KUKA KRL program: MyProgram_206().src

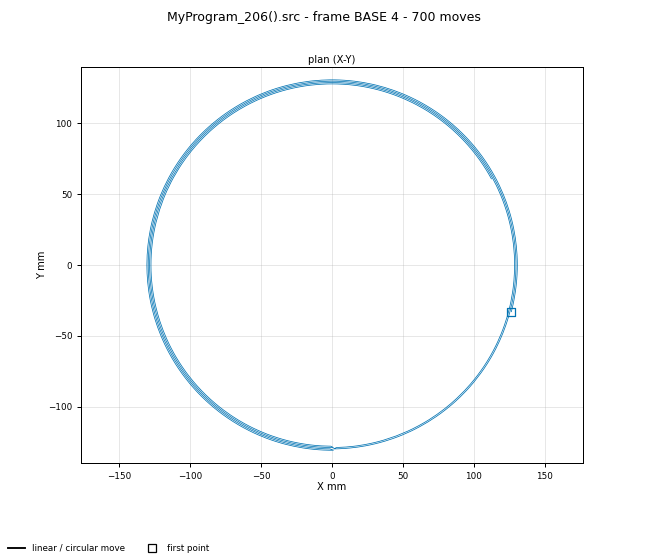
[picture p0: tool path of MyProgram_206().src in frame BASE 4, 700 of 700 moves have a stored position in this frame; points joined in program order, loops and branches not executed]
&ACCESS RVP
&REL 1
&PARAM TEMPLATE = C:\KRC\Roboter\Template\vorgabe
&PARAM EDITMASK = *
DEF MyProgram_206()
; ---- Setting reference (Base) ----
$BASE = BASE_DATA[4]

; --------------------------
; ---- Setting tool (TCP) ----
$TOOL = TOOL_DATA[3]
; --------------------------

$VEL.CP = VEL_APROX_PRINT
Startdeposition()
$VEL.CP = VEL_PRINT
LIN {X 126.4468,Y -32.9033,Z 147,A -17.6105,B 24.9579,C -1.4995,E1 25.155,E2 463.9583} C_DIS
LIN {X 127.5485,Y -28.3334,Z 147,A -15.6439,B 24.9578,C -1.501,E1 25.1563,E2 461.9995} C_DIS
LIN {X 128.2452,Y -24.9837,Z 147,A -14.1957,B 24.9577,C -1.5031,E1 25.1571,E2 460.5549} C_DIS
LIN {X 128.8355,Y -21.7323,Z 147,A -12.7991,B 24.9576,C -1.505,E1 25.1577,E2 459.162} C_DIS
LIN {X 129.3075,Y -18.7203,Z 147,A -11.4837,B 24.9574,C -1.5082,E1 25.1583,E2 457.8467} C_DIS
LIN {X 129.825,Y -14.7267,Z 147,A -9.5964,B 24.9567,C -1.5207,E1 25.1589,E2 455.9413} C_DIS
LIN {X 130.2553,Y -10.2444,Z 147,A -7.7715,B 24.9567,C -1.519,E1 25.1594,E2 454.1311} C_DIS
LIN {X 130.4729,Y -6.9157,Z 147,A -6.2379,B 24.9563,C -1.5277,E1 25.1596,E2 452.586} C_DIS
LIN {X 130.6151,Y -3.2719,Z 147,A -4.7193,B 24.9563,C -1.5286,E1 25.1598,E2 451.0743} C_DIS
LIN {X 130.6591,Y 0,Z 147,A -3.1934,B 24.9557,C -1.5383,E1 25.1598,E2 449.5347} C_DIS
LIN {X 130.6081,Y 3.5243,Z 147,A -1.7202,B 24.9556,C -1.5395,E1 25.1597,E2 448.0675} C_DIS
LIN {X 130.4538,Y 7.2957,Z 147,A 0.0234,B 24.955,C -1.5497,E1 25.1595,E2 446.3101} C_DIS
LIN {X 130.1886,Y 11.036,Z 147,A 1.3411,B 24.9557,C -1.5373,E1 25.1592,E2 445.0295} C_DIS
LIN {X 129.9628,Y 13.4458,Z 147,A 2.6602,B 24.9547,C -1.5548,E1 25.1588,E2 443.6769} C_DIS
LIN {X 129.6461,Y 16.2263,Z 147,A 3.8628,B 24.9546,C -1.5574,E1 25.1584,E2 442.4753} C_DIS
LIN {X 129.2338,Y 19.2365,Z 147,A 5.1142,B 24.9546,C -1.5574,E1 25.1579,E2 441.2315} C_DIS
LIN {X 128.6452,Y 22.8309,Z 147,A 6.4775,B 24.955,C -1.5498,E1 25.1573,E2 439.8941} C_DIS
LIN {X 128.1418,Y 25.5106,Z 147,A 7.8931,B 24.9541,C -1.5656,E1 25.1565,E2 438.4495} C_DIS
LIN {X 127.5485,Y 28.3334,Z 147,A 9.2267,B 24.9536,C -1.5733,E1 25.1557,E2 437.1054} C_DIS
LIN {X 126.7277,Y 31.7964,Z 147,A 10.7556,B 24.9534,C -1.5765,E1 25.1547,E2 435.5777} C_DIS
LIN {X 125.9076,Y 34.9019,Z 147,A 12.104,B 24.9534,C -1.5777,E1 25.1537,E2 434.2343} C_DIS
LIN {X 124.9889,Y 38.0602,Z 147,A 13.541,B 24.9531,C -1.5819,E1 25.1526,E2 432.7957} C_DIS
LIN {X 123.9957,Y 41.1807,Z 147,A 14.8652,B 24.9532,C -1.5802,E1 25.1515,E2 431.4829} C_DIS
LIN {X 122.993,Y 44.0856,Z 147,A 16.2938,B 24.9527,C -1.5887,E1 25.1501,E2 430.0423} C_DIS
LIN {X 121.8877,Y 47.0557,Z 147,A 17.4959,B 24.9531,C -1.5827,E1 25.149,E2 428.861} C_DIS
LIN {X 120.8768,Y 49.6004,Z 147,A 18.8871,B 24.9522,C -1.5966,E1 25.1475,E2 427.4448} C_DIS
LIN {X 119.4073,Y 53.0353,Z 147,A 20.3317,B 24.9526,C -1.5909,E1 25.1459,E2 426.0214} C_DIS
LIN {X 118.1445,Y 55.7938,Z 147,A 21.9257,B 24.9515,C -1.6091,E1 25.144,E2 424.3933} C_DIS
LIN {X 116.5299,Y 59.0893,Z 147,A 23.3217,B 24.9519,C -1.6022,E1 25.1423,E2 423.021} C_DIS
LIN {X 114.9008,Y 62.2029,Z 147,A 25.1201,B 24.9508,C -1.6204,E1 25.1399,E2 421.1891} C_DIS
LIN {X 112.8073,Y 65.923,Z 147,A 26.8375,B 24.951,C -1.6172,E1 25.1375,E2 419.4881} C_DIS
LIN {X 110.7749,Y 69.2838,Z 147,A 28.6456,B 24.9504,C -1.6265,E1 25.1348,E2 417.6673} C_DIS
LIN {X 108.4346,Y 72.8927,Z 147,A 30.56,B 24.95,C -1.633,E1 25.1319,E2 415.7472} C_DIS
LIN {X 105.9386,Y 76.4742,Z 147,A 32.4107,B 24.95,C -1.6345,E1 25.1289,E2 413.9019} C_DIS
LIN {X 103.4746,Y 79.7768,Z 147,A 34.2161,B 24.9497,C -1.6389,E1 25.1258,E2 412.0946} C_DIS
LIN {X 100.8929,Y 83.0182,Z 147,A 36.0737,B 24.9493,C -1.6455,E1 25.1226,E2 410.2301} C_DIS
LIN {X 97.9836,Y 86.4318,Z 147,A 37.9938,B 24.9491,C -1.6476,E1 25.1191,E2 408.3137} C_DIS
LIN {X 94.9376,Y 89.767,Z 147,A 39.9231,B 24.9491,C -1.6494,E1 25.1154,E2 406.3886} C_DIS
LIN {X 91.9122,Y 92.8625,Z 147,A 41.8417,B 24.9487,C -1.6547,E1 25.1116,E2 404.4657} C_DIS
LIN {X 88.7329,Y 95.9056,Z 147,A 43.8155,B 24.9483,C -1.6611,E1 25.1076,E2 402.485} C_DIS
LIN {X 85.5245,Y 98.777,Z 147,A 45.651,B 24.9483,C -1.6621,E1 25.1037,E2 400.6542} C_DIS
LIN {X 82.3328,Y 101.4529,Z 147,A 47.4623,B 24.9481,C -1.6649,E1 25.0998,E2 398.8434} C_DIS
LIN {X 79.0403,Y 104.0387,Z 147,A 49.2387,B 24.9481,C -1.6651,E1 25.0959,E2 397.0729} C_DIS
LIN {X 76.2379,Y 106.109,Z 147,A 50.8439,B 24.9476,C -1.6719,E1 25.0923,E2 395.4573} C_DIS
LIN {X 72.8927,Y 108.4346,Z 147,A 52.6181,B 24.9475,C -1.6743,E1 25.0882,E2 393.6835} C_DIS
LIN {X 69.2662,Y 110.7858,Z 147,A 54.5215,B 24.9473,C -1.6778,E1 25.0837,E2 391.778} C_DIS
LIN {X 65.2644,Y 113.1894,Z 147,A 56.5241,B 24.9473,C -1.6785,E1 25.0789,E2 389.7798} C_DIS
LIN {X 61.4738,Y 115.2926,Z 147,A 58.3276,B 24.9473,C -1.676,E1 25.0745,E2 387.9873} C_DIS
LIN {X 58.5401,Y 116.8095,Z 147,A 59.7705,B 24.9473,C -1.6777,E1 25.0709,E2 386.5445} C_DIS
LIN {X 55.1242,Y 118.4574,Z 147,A 61.4114,B 24.9472,C -1.6786,E1 25.0668,E2 384.9056} C_DIS
LIN {X 52.3074,Y 119.7285,Z 147,A 62.8038,B 24.947,C -1.6821,E1 25.0632,E2 383.5084} C_DIS
LIN {X 49.2079,Y 121.0351,Z 147,A 64.186,B 24.9472,C -1.6789,E1 25.0597,E2 382.1371} C_DIS
LIN {X 46.0827,Y 122.2588,Z 147,A 65.7194,B 24.9469,C -1.6835,E1 25.0557,E2 380.5959} C_DIS
LIN {X 43.1226,Y 123.3342,Z 147,A 67.0966,B 24.9469,C -1.6846,E1 25.052,E2 379.2191} C_DIS
LIN {X 40.044,Y 124.3678,Z 147,A 68.3559,B 24.9473,C -1.6773,E1 25.0487,E2 377.9794} C_DIS
LIN {X 37.0878,Y 125.2814,Z 147,A 69.887,B 24.9466,C -1.6873,E1 25.0446,E2 376.4274} C_DIS
LIN {X 34.0705,Y 126.1355,Z 147,A 71.0918,B 24.9471,C -1.6795,E1 25.0414,E2 375.243} C_DIS
LIN {X 31.1608,Y 126.8862,Z 147,A 72.5499,B 24.9466,C -1.6875,E1 25.0374,E2 373.7681} C_DIS
LIN {X 28.3334,Y 127.5485,Z 147,A 73.8201,B 24.9466,C -1.688,E1 25.034,E2 372.4985} C_DIS
LIN {X 24.8107,Y 128.2783,Z 147,A 75.2022,B 24.9472,C -1.6788,E1 25.0302,E2 371.14} C_DIS
LIN {X 22.0424,Y 128.7837,Z 147,A 76.6946,B 24.9463,C -1.6924,E1 25.0261,E2 369.6168} C_DIS
LIN {X 18.5992,Y 129.3248,Z 147,A 78.0161,B 24.947,C -1.6823,E1 25.0225,E2 368.3205} C_DIS
LIN {X 16.0112,Y 129.6718,Z 147,A 79.4052,B 24.9462,C -1.695,E1 25.0185,E2 366.9024} C_DIS
LIN {X 12.5076,Y 130.0554,Z 147,A 80.7941,B 24.9467,C -1.6873,E1 25.0147,E2 365.5328} C_DIS
LIN {X 8.7721,Y 130.3628,Z 147,A 82.547,B 24.9463,C -1.6929,E1 25.0098,E2 363.7675} C_DIS
LIN {X 5.3158,Y 130.5476,Z 147,A 84.0144,B 24.9465,C -1.6903,E1 25.0057,E2 362.3067} C_DIS
LIN {X 1.9502,Y 130.6412,Z 147,A 85.5842,B 24.9462,C -1.6948,E1 25.0013,E2 360.7264} C_DIS
LIN {X -1.6553,Y 130.6461,Z 147,A 86.9652,B 24.9468,C -1.6844,E1 24.9975,E2 359.3702} C_DIS
LIN {X -4.8429,Y 130.566,Z 147,A 88.5082,B 24.9464,C -1.6912,E1 24.9932,E2 357.8106} C_DIS
LIN {X -7.5075,Y 130.4407,Z 147,A 89.6225,B 24.9466,C -1.688,E1 24.9901,E2 356.7037} C_DIS
LIN {X -10.6813,Y 130.2185,Z 147,A 91.0433,B 24.9466,C -1.6887,E1 24.9861,E2 355.2807} C_DIS
LIN {X -13.7959,Y 129.9252,Z 147,A 92.2181,B 24.9472,C -1.6781,E1 24.983,E2 354.1304} C_DIS
LIN {X -16.2263,Y 129.6461,Z 147,A 93.5478,B 24.9465,C -1.6903,E1 24.9792,E2 352.7708} C_DIS
LIN {X -19.7661,Y 129.1518,Z 147,A 94.9747,B 24.947,C -1.6823,E1 24.9753,E2 351.3619} C_DIS
LIN {X -22.4768,Y 128.7086,Z 147,A 96.167,B 24.947,C -1.6807,E1 24.972,E2 350.172} C_DIS
LIN {X -25.5106,Y 128.1418,Z 147,A 97.6901,B 24.9466,C -1.6881,E1 24.9678,E2 348.6298} C_DIS
LIN {X -28.8224,Y 127.4368,Z 147,A 99.0733,B 24.947,C -1.6817,E1 24.964,E2 347.26} C_DIS
LIN {X -31.879,Y 126.7067,Z 147,A 100.4803,B 24.947,C -1.6817,E1 24.9602,E2 345.8508} C_DIS
LIN {X -34.9823,Y 125.8851,Z 147,A 101.9129,B 24.947,C -1.6816,E1 24.9564,E2 344.4166} C_DIS
LIN {X -38.9977,Y 124.702,Z 147,A 103.8195,B 24.947,C -1.6829,E1 24.9512,E2 342.5036} C_DIS
LIN {X -42.0389,Y 123.7099,Z 147,A 105.2281,B 24.947,C -1.6815,E1 24.9475,E2 341.0957} C_DIS
LIN {X -45.0722,Y 122.6373,Z 147,A 106.5653,B 24.9474,C -1.676,E1 24.944,E2 339.7688} C_DIS
LIN {X -48.561,Y 121.2958,Z 147,A 108.0134,B 24.9481,C -1.6644,E1 24.9403,E2 338.3453} C_DIS
LIN {X -51.1024,Y 120.2495,Z 147,A 109.5022,B 24.9473,C -1.6765,E1 24.9364,E2 336.8242} C_DIS
LIN {X -54.3102,Y 118.8338,Z 147,A 111.0526,B 24.9474,C -1.6748,E1 24.9325,E2 335.2741} C_DIS
LIN {X -57.4981,Y 117.3235,Z 147,A 112.4977,B 24.9479,C -1.6673,E1 24.9289,E2 333.843} C_DIS
LIN {X -60.2203,Y 115.9508,Z 147,A 113.9489,B 24.9477,C -1.6707,E1 24.9252,E2 332.38} C_DIS
LIN {X -64.2753,Y 113.7541,Z 147,A 115.9667,B 24.9479,C -1.6669,E1 24.9203,E2 330.3655} C_DIS
LIN {X -67.9659,Y 111.5887,Z 147,A 117.913,B 24.9479,C -1.6668,E1 24.9156,E2 328.4133} C_DIS
LIN {X -71.6939,Y 109.2303,Z 147,A 119.8293,B 24.9482,C -1.6621,E1 24.9111,E2 326.5019} C_DIS
LIN {X -74.9667,Y 107.0113,Z 147,A 121.4987,B 24.9486,C -1.6554,E1 24.9073,E2 324.8428} C_DIS
LIN {X -77.7906,Y 104.9759,Z 147,A 122.9997,B 24.9489,C -1.651,E1 24.904,E2 323.3471} C_DIS
LIN {X -80.9423,Y 102.5654,Z 147,A 124.8156,B 24.9489,C -1.6509,E1 24.8999,E2 321.5248} C_DIS
LIN {X -84.3028,Y 99.822,Z 147,A 126.6937,B 24.9493,C -1.6454,E1 24.8959,E2 319.6525} C_DIS
LIN {X -87.3944,Y 97.1264,Z 147,A 128.4827,B 24.9496,C -1.6408,E1 24.8922,E2 317.8676} C_DIS
LIN {X -90.0542,Y 94.6655,Z 147,A 130.1941,B 24.9494,C -1.6428,E1 24.8887,E2 316.1442} C_DIS
LIN {X -93.0698,Y 91.7024,Z 147,A 132.0482,B 24.9497,C -1.6383,E1 24.885,E2 314.2932} C_DIS
LIN {X -95.9056,Y 88.7329,Z 147,A 133.866,B 24.9499,C -1.6345,E1 24.8816,E2 312.4763} C_DIS
LIN {X -98.7242,Y 85.5859,Z 147,A 135.7281,B 24.9502,C -1.6301,E1 24.8781,E2 310.6162} C_DIS
LIN {X -101.4364,Y 82.3532,Z 147,A 137.5974,B 24.9505,C -1.6261,E1 24.8748,E2 308.7479} C_DIS
LIN {X -104.1842,Y 78.8474,Z 147,A 139.5324,B 24.9508,C -1.6199,E1 24.8715,E2 306.8185} C_DIS
LIN {X -106.8115,Y 75.2499,Z 147,A 141.446,B 24.9513,C -1.6125,E1 24.8684,E2 304.913} C_DIS
LIN {X -108.9656,Y 72.0959,Z 147,A 143.1927,B 24.9513,C -1.6112,E1 24.8657,E2 303.1609} C_DIS
LIN {X -111.2152,Y 68.5748,Z 147,A 144.9176,B 24.952,C -1.6007,E1 24.8632,E2 301.452} C_DIS
LIN {X -113.2245,Y 65.2038,Z 147,A 146.7184,B 24.952,C -1.5995,E1 24.8606,E2 299.645} C_DIS
LIN {X -115.2926,Y 61.4738,Z 147,A 148.675,B 24.9522,C -1.598,E1 24.858,E2 297.6815} C_DIS
LIN {X -117.0096,Y 58.1346,Z 147,A 150.0067,B 24.9533,C -1.5781,E1 24.8564,E2 296.3902} C_DIS
LIN {X -118.3448,Y 55.3678,Z 147,A 151.575,B 24.953,C -1.5844,E1 24.8545,E2 294.7982} C_DIS
LIN {X -119.7487,Y 52.2607,Z 147,A 153.0994,B 24.9532,C -1.5812,E1 24.8527,E2 293.2731} C_DIS
LIN {X -120.9639,Y 49.3844,Z 147,A 154.4694,B 24.9534,C -1.5769,E1 24.8513,E2 291.9057} C_DIS
LIN {X -122.2722,Y 46.0468,Z 147,A 155.9491,B 24.954,C -1.5676,E1 24.8498,E2 290.4398} C_DIS
LIN {X -123.3462,Y 43.0879,Z 147,A 157.4104,B 24.954,C -1.5671,E1 24.8484,E2 288.9716} C_DIS
LIN {X -124.4183,Y 39.8858,Z 147,A 158.796,B 24.9545,C -1.5578,E1 24.8472,E2 287.6001} C_DIS
LIN {X -125.319,Y 36.9594,Z 147,A 160.0163,B 24.9551,C -1.5477,E1 24.8463,E2 286.3969} C_DIS
LIN {X -126.1631,Y 33.9669,Z 147,A 161.5501,B 24.9549,C -1.5514,E1 24.8451,E2 284.8454} C_DIS
LIN {X -126.9441,Y 30.9205,Z 147,A 162.9045,B 24.9552,C -1.5457,E1 24.8442,E2 283.4966} C_DIS
LIN {X -127.5485,Y 28.3334,Z 147,A 164.1567,B 24.9552,C -1.546,E1 24.8434,E2 282.2364} C_DIS
LIN {X -128.2278,Y 25.0749,Z 147,A 165.5371,B 24.9557,C -1.5375,E1 24.8426,E2 280.8681} C_DIS
LIN {X -128.8216,Y 21.8154,Z 147,A 167.1088,B 24.9557,C -1.5384,E1 24.8419,E2 279.285} C_DIS
LIN {X -129.3132,Y 18.6808,Z 147,A 168.4212,B 24.9561,C -1.5301,E1 24.8413,E2 277.9845} C_DIS
LIN {X -129.6718,Y 16.0112,Z 147,A 169.5862,B 24.9564,C -1.5254,E1 24.8409,E2 276.8238} C_DIS
LIN {X -129.9859,Y 13.2313,Z 147,A 170.978,B 24.9562,C -1.5291,E1 24.8405,E2 275.4146} C_DIS
LIN {X -130.2546,Y 10.2537,Z 147,A 172.2222,B 24.9566,C -1.5216,E1 24.8402,E2 274.1808} C_DIS
LIN {X -130.4644,Y 7.0847,Z 147,A 173.7111,B 24.9566,C -1.5216,E1 24.84,E2 272.683} C_DIS
LIN {X -130.6254,Y 2.9001,Z 147,A 175.5599,B 24.9569,C -1.5161,E1 24.8398,E2 270.8362} C_DIS
LIN {X -130.6591,Y 0,Z 147,A 176.8654,B 24.9571,C -1.5135,E1 24.8398,E2 269.5291} C_DIS
LIN {X -130.6254,Y -2.9001,Z 147,A 178.1031,B 24.9574,C -1.5077,E1 24.8398,E2 268.2978} C_DIS
LIN {X -130.5277,Y -5.8247,Z 147,A 179.493,B 24.9574,C -1.5086,E1 24.84,E2 266.8974} C_DIS
LIN {X -130.3473,Y -8.9846,Z 147,A -179.3585,B 24.9583,C -1.4927,E1 24.8402,E2 265.7799} C_DIS
LIN {X -130.1086,Y -11.954,Z 147,A -177.8743,B 24.958,C -1.4968,E1 24.8406,E2 264.2769} C_DIS
LIN {X -129.7374,Y -15.4615,Z 147,A -176.4479,B 24.9586,C -1.4861,E1 24.841,E2 262.8675} C_DIS
LIN {X -129.3449,Y -18.4591,Z 147,A -175.0501,B 24.9586,C -1.4853,E1 24.8415,E2 261.4633} C_DIS
LIN {X -128.8678,Y -21.5388,Z 147,A -173.6499,B 24.9588,C -1.4824,E1 24.8422,E2 260.0616} C_DIS
LIN {X -128.1862,Y -25.2926,Z 147,A -171.8404,B 24.9588,C -1.4836,E1 24.8431,E2 258.2387} C_DIS
LIN {X -127.3992,Y -28.987,Z 147,A -170.3065,B 24.9594,C -1.4725,E1 24.844,E2 256.7221} C_DIS
LIN {X -126.6514,Y -32.0972,Z 147,A -168.9134,B 24.9596,C -1.4676,E1 24.845,E2 255.3324} C_DIS
LIN {X -125.8807,Y -34.9982,Z 147,A -167.5943,B 24.9599,C -1.4637,E1 24.8459,E2 254.0151} C_DIS
LIN {X -125.0295,Y -37.9276,Z 147,A -166.2896,B 24.9602,C -1.4579,E1 24.847,E2 252.7166} C_DIS
LIN {X -124.0468,Y -41.0273,Z 147,A -165.0073,B 24.9608,C -1.4467,E1 24.8481,E2 251.4537} C_DIS
LIN {X -123.0459,Y -43.9388,Z 147,A -163.4254,B 24.9604,C -1.4536,E1 24.8495,E2 249.8462} C_DIS
LIN {X -121.8557,Y -47.1379,Z 147,A -162.1612,B 24.9613,C -1.438,E1 24.8507,E2 248.6122} C_DIS
LIN {X -120.698,Y -50.0285,Z 147,A -160.5232,B 24.9608,C -1.447,E1 24.8525,E2 246.9436} C_DIS
LIN {X -119.4912,Y -52.8477,Z 147,A -159.1822,B 24.961,C -1.4429,E1 24.854,E2 245.6051} C_DIS
LIN {X -118.0955,Y -55.8965,Z 147,A -157.7431,B 24.9613,C -1.4371,E1 24.8557,E2 244.1719} C_DIS
LIN {X -116.6819,Y -58.7907,Z 147,A -156.3083,B 24.9615,C -1.4341,E1 24.8575,E2 242.7364} C_DIS
LIN {X -114.9008,Y -62.2029,Z 147,A -154.447,B 24.9613,C -1.4377,E1 24.8599,E2 240.8567} C_DIS
LIN {X -112.796,Y -65.9422,Z 147,A -152.5718,B 24.9616,C -1.4323,E1 24.8625,E2 238.9847} C_DIS
LIN {X -110.4716,Y -69.7658,Z 147,A -150.6656,B 24.962,C -1.4243,E1 24.8653,E2 237.0878} C_DIS
LIN {X -108.209,Y -73.226,Z 147,A -148.8313,B 24.9622,C -1.4206,E1 24.8682,E2 235.2532} C_DIS
LIN {X -105.7592,Y -76.7218,Z 147,A -146.9627,B 24.9625,C -1.4156,E1 24.8712,E2 233.3872} C_DIS
LIN {X -103.2394,Y -80.0804,Z 147,A -145.0767,B 24.9625,C -1.4132,E1 24.8744,E2 231.4979} C_DIS
LIN {X -100.4417,Y -83.563,Z 147,A -143.1001,B 24.9628,C -1.4093,E1 24.8779,E2 229.5214} C_DIS
LIN {X -97.6093,Y -86.8553,Z 147,A -141.2483,B 24.9632,C -1.4023,E1 24.8813,E2 227.678} C_DIS
LIN {X -94.8325,Y -89.8783,Z 147,A -139.4585,B 24.9634,C -1.3977,E1 24.8847,E2 225.8912} C_DIS
LIN {X -92.3028,Y -92.4744,Z 147,A -137.7574,B 24.9633,C -1.3997,E1 24.888,E2 224.1781} C_DIS
LIN {X -89.2184,Y -95.4534,Z 147,A -135.9108,B 24.9636,C -1.3941,E1 24.8918,E2 222.3372} C_DIS
LIN {X -86.164,Y -98.2197,Z 147,A -134.0432,B 24.9636,C -1.3934,E1 24.8957,E2 220.4638} C_DIS
LIN {X -82.9751,Y -100.9283,Z 147,A -132.2676,B 24.964,C -1.387,E1 24.8995,E2 218.6969} C_DIS
LIN {X -79.709,Y -103.5272,Z 147,A -130.4002,B 24.964,C -1.3854,E1 24.9036,E2 216.8263} C_DIS
LIN {X -76.3359,Y -106.0389,Z 147,A -128.643,B 24.9644,C -1.3778,E1 24.9075,E2 215.0809} C_DIS
LIN {X -73.2555,Y -108.1891,Z 147,A -126.9211,B 24.9644,C -1.3788,E1 24.9115,E2 213.351} C_DIS
LIN {X -69.6535,Y -110.5424,Z 147,A -125.0525,B 24.9646,C -1.3749,E1 24.9159,E2 211.4857} C_DIS
LIN {X -65.9714,Y -112.7788,Z 147,A -123.15,B 24.9647,C -1.3727,E1 24.9204,E2 209.5825} C_DIS
LIN {X -62.2029,Y -114.9008,Z 147,A -121.159,B 24.9646,C -1.3748,E1 24.9253,E2 207.5809} C_DIS
LIN {X -58.2704,Y -116.9426,Z 147,A -119.328,B 24.965,C -1.3667,E1 24.9299,E2 205.7642} C_DIS
LIN {X -55.3678,Y -118.3448,Z 147,A -117.8647,B 24.965,C -1.3675,E1 24.9336,E2 204.2952} C_DIS
LIN {X -52.2698,Y -119.7448,Z 147,A -116.4901,B 24.9654,C -1.3599,E1 24.937,E2 202.9352} C_DIS
LIN {X -49.2658,Y -121.0117,Z 147,A -115.0159,B 24.9654,C -1.3607,E1 24.9408,E2 201.4559} C_DIS
LIN {X -46.342,Y -122.1617,Z 147,A -113.6372,B 24.9654,C -1.3594,E1 24.9444,E2 200.0773} C_DIS
LIN {X -43.3007,Y -123.2725,Z 147,A -112.2465,B 24.9655,C -1.3566,E1 24.9481,E2 198.6904} C_DIS
LIN {X -40.0328,Y -124.3713,Z 147,A -110.6692,B 24.9655,C -1.3587,E1 24.9523,E2 197.1052} C_DIS
LIN {X -35.9515,Y -125.6141,Z 147,A -108.8335,B 24.9655,C -1.3556,E1 24.9572,E2 195.274} C_DIS
LIN {X -32.9033,Y -126.4468,Z 147,A -107.3711,B 24.9655,C -1.3586,E1 24.9612,E2 193.8022} C_DIS
LIN {X -29.6375,Y -127.2506,Z 147,A -105.8847,B 24.9655,C -1.3584,E1 24.9652,E2 192.3142} C_DIS
LIN {X -26.8122,Y -127.8769,Z 147,A -104.6293,B 24.9655,C -1.3571,E1 24.9686,E2 191.0604} C_DIS
LIN {X -23.1695,Y -128.5847,Z 147,A -103.092,B 24.9658,C -1.3519,E1 24.9728,E2 189.5337} C_DIS
LIN {X -20.5299,Y -129.0335,Z 147,A -101.8286,B 24.9656,C -1.3561,E1 24.9763,E2 188.2593} C_DIS
LIN {X -17.1528,Y -129.5247,Z 147,A -100.3973,B 24.9657,C -1.3525,E1 24.9803,E2 186.8355} C_DIS
LIN {X -13.2313,Y -129.9859,Z 147,A -98.6095,B 24.9657,C -1.3551,E1 24.9853,E2 185.0404} C_DIS
LIN {X -9.835,Y -130.2852,Z 147,A -97.1159,B 24.9657,C -1.355,E1 24.9894,E2 183.5464} C_DIS
LIN {X -6.2891,Y -130.5044,Z 147,A -95.523,B 24.9655,C -1.3569,E1 24.9939,E2 181.9485} C_DIS
LIN {X -2.2444,Y -130.6363,Z 147,A -93.892,B 24.9659,C -1.3497,E1 24.9984,E2 180.3343} C_DIS
LIN {X 0.9279,Y -130.6497,Z 147,A -92.6871,B 24.9663,C -1.3405,E1 25.0017,E2 179.1513} C_DIS
Enddeposition()
LIN {X 0.9279,Y -130.6497,Z 147,A -92.6871,B 24.9663,C -1.3405,E1 25.0017,E2 179.1513} C_DIS
Startdeposition()
$VEL.CP = VEL_PRINT
LIN {X -1.4285,Y -129.6952,Z 147,A -93.99,B 24.0899,C -1.1624,E1 24.1134,E2 180.7672} C_DIS
LIN {X -5.453,Y -129.587,Z 147,A -95.623,B 24.0896,C -1.1693,E1 24.1089,E2 182.3836} C_DIS
LIN {X -9.475,Y -129.3544,Z 147,A -97.4578,B 24.0897,C -1.1666,E1 24.1038,E2 184.2257} C_DIS
LIN {X -14.5615,Y -128.8828,Z 147,A -99.7879,B 24.0899,C -1.1632,E1 24.0973,E2 186.5654} C_DIS
LIN {X -18.0218,Y -128.4432,Z 147,A -101.481,B 24.0902,C -1.1563,E1 24.0925,E2 188.2769} C_DIS
LIN {X -21.676,Y -127.8772,Z 147,A -103.4016,B 24.0908,C -1.143,E1 24.0872,E2 190.2319} C_DIS
LIN {X -26.0272,Y -127.0626,Z 147,A -104.8454,B 24.0896,C -1.1683,E1 24.0834,E2 191.6153} C_DIS
LIN {X -29.9496,Y -126.1963,Z 147,A -106.6062,B 24.0896,C -1.1699,E1 24.0786,E2 193.3747} C_DIS
LIN {X -32.8253,Y -125.4797,Z 147,A -107.81,B 24.0893,C -1.1757,E1 24.0753,E2 194.5661} C_DIS
LIN {X -35.9455,Y -124.6213,Z 147,A -109.3552,B 24.0895,C -1.1711,E1 24.0711,E2 196.125} C_DIS
LIN {X -39.2637,Y -123.615,Z 147,A -110.964,B 24.0896,C -1.1686,E1 24.0668,E2 197.7428} C_DIS
LIN {X -43.626,Y -122.1441,Z 147,A -112.9166,B 24.0894,C -1.1742,E1 24.0617,E2 199.6857} C_DIS
LIN {X -46.9487,Y -120.9052,Z 147,A -114.4528,B 24.0892,C -1.1771,E1 24.0577,E2 201.218} C_DIS
LIN {X -49.4552,Y -119.9029,Z 147,A -115.7583,B 24.0894,C -1.173,E1 24.0543,E2 202.5367} C_DIS
LIN {X -52.5326,Y -118.5866,Z 147,A -117.4165,B 24.0897,C -1.1662,E1 24.05,E2 204.2159} C_DIS
LIN {X -57.1398,Y -116.436,Z 147,A -119.4068,B 24.089,C -1.1809,E1 24.0451,E2 206.1751} C_DIS
LIN {X -60.1065,Y -114.9325,Z 147,A -120.8902,B 24.089,C -1.1822,E1 24.0414,E2 207.6597} C_DIS
LIN {X -63.8439,Y -112.9017,Z 147,A -122.8788,B 24.0891,C -1.1796,E1 24.0365,E2 209.6606} C_DIS
LIN {X -66.7959,Y -111.1808,Z 147,A -124.4146,B 24.0891,C -1.1806,E1 24.0328,E2 211.1988} C_DIS
LIN {X -69.9805,Y -109.2038,Z 147,A -126.0465,B 24.0889,C -1.1843,E1 24.029,E2 212.827} C_DIS
LIN {X -73.6101,Y -106.7912,Z 147,A -128.1124,B 24.089,C -1.1809,E1 24.0241,E2 214.9084} C_DIS
LIN {X -77.7054,Y -103.8494,Z 147,A -130.1925,B 24.0885,C -1.1917,E1 24.0195,E2 216.9697} C_DIS
LIN {X -81.0145,Y -101.289,Z 147,A -132.0596,B 24.0885,C -1.1942,E1 24.0154,E2 218.8378} C_DIS
LIN {X -84.2468,Y -98.6169,Z 147,A -133.9299,B 24.0883,C -1.197,E1 24.0114,E2 220.7087} C_DIS
LIN {X -87.488,Y -95.7535,Z 147,A -135.8702,B 24.0882,C -1.1995,E1 24.0074,E2 222.6509} C_DIS
LIN {X -90.5463,Y -92.8667,Z 147,A -137.6775,B 24.0879,C -1.2057,E1 24.0037,E2 224.4508} C_DIS
LIN {X -93.4992,Y -89.8931,Z 147,A -139.6002,B 24.0879,C -1.2065,E1 24,E2 226.3802} C_DIS
LIN {X -96.5557,Y -86.6009,Z 147,A -141.5588,B 24.0876,C -1.2122,E1 23.9963,E2 228.3337} C_DIS
LIN {X -99.5375,Y -83.1569,Z 147,A -143.564,B 24.0873,C -1.2172,E1 23.9927,E2 230.3361} C_DIS
LIN {X -101.5973,Y -80.6272,Z 147,A -145.093,B 24.0873,C -1.2167,E1 23.99,E2 231.8739} C_DIS
LIN {X -104.2928,Y -77.1096,Z 147,A -146.9906,B 24.087,C -1.2242,E1 23.9868,E2 233.7623} C_DIS
LIN {X -106.6795,Y -73.7722,Z 147,A -148.8378,B 24.0869,C -1.2273,E1 23.9838,E2 235.6115} C_DIS
LIN {X -109.0442,Y -70.2297,Z 147,A -150.7243,B 24.0866,C -1.232,E1 23.981,E2 237.4963} C_DIS
LIN {X -111.2632,Y -66.6582,Z 147,A -152.3298,B 24.0858,C -1.2484,E1 23.9787,E2 239.0699} C_DIS
LIN {X -112.93,Y -63.7937,Z 147,A -154.0799,B 24.0863,C -1.2394,E1 23.9762,E2 240.8516} C_DIS
LIN {X -115.4539,Y -59.0992,Z 147,A -156.3342,B 24.0857,C -1.2505,E1 23.9733,E2 243.0911} C_DIS
LIN {X -116.9467,Y -56.0868,Z 147,A -157.8188,B 24.0855,C -1.2548,E1 23.9714,E2 244.5735} C_DIS
LIN {X -118.3456,Y -53.0714,Z 147,A -159.3067,B 24.0854,C -1.2581,E1 23.9697,E2 246.0616} C_DIS
LIN {X -119.7306,Y -49.8681,Z 147,A -160.801,B 24.085,C -1.2648,E1 23.9681,E2 247.5482} C_DIS
LIN {X -121.7133,Y -44.8178,Z 147,A -163.7609,B 24.0859,C -1.2466,E1 23.9651,E2 250.5702} C_DIS
LIN {X -123.0532,Y -40.99,Z 147,A -165.0397,B 24.0845,C -1.275,E1 23.964,E2 251.7866} C_DIS
LIN {X -124.0511,Y -37.863,Z 147,A -166.5279,B 24.0844,C -1.2777,E1 23.9628,E2 253.2771} C_DIS
LIN {X -125.0653,Y -34.3699,Z 147,A -168.1434,B 24.0842,C -1.2823,E1 23.9615,E2 254.8911} C_DIS
LIN {X -126.0168,Y -30.6943,Z 147,A -169.8527,B 24.084,C -1.2861,E1 23.9604,E2 256.6014} C_DIS
LIN {X -126.7877,Y -27.3344,Z 147,A -171.3695,B 24.0837,C -1.2911,E1 23.9594,E2 258.115} C_DIS
LIN {X -127.5438,Y -23.5672,Z 147,A -173.1992,B 24.0837,C -1.2905,E1 23.9585,E2 259.9575} C_DIS
LIN {X -128.1733,Y -19.8474,Z 147,A -174.8005,B 24.0833,C -1.2988,E1 23.9578,E2 261.5483} C_DIS
LIN {X -128.7579,Y -15.6138,Z 147,A -176.6653,B 24.083,C -1.3059,E1 23.9571,E2 263.4073} C_DIS
LIN {X -129.1188,Y -12.276,Z 147,A -178.1607,B 24.0828,C -1.3101,E1 23.9567,E2 264.9016} C_DIS
LIN {X -129.4407,Y -8.2168,Z 147,A -179.9871,B 24.0825,C -1.3147,E1 23.9563,E2 266.7281} C_DIS
LIN {X -129.6132,Y -4.7812,Z 147,A 178.445,B 24.0824,C -1.3175,E1 23.9561,E2 268.2989} C_DIS
LIN {X -129.6982,Y -1.0161,Z 147,A 176.7931,B 24.0821,C -1.3234,E1 23.9561,E2 269.9466} C_DIS
LIN {X -129.6668,Y 3.0361,Z 147,A 174.955,B 24.0819,C -1.3271,E1 23.9561,E2 271.787} C_DIS
LIN {X -129.5261,Y 6.7384,Z 147,A 173.3981,B 24.0814,C -1.3361,E1 23.9563,E2 273.3317} C_DIS
LIN {X -129.266,Y 10.6172,Z 147,A 171.6128,B 24.0813,C -1.3386,E1 23.9567,E2 275.1218} C_DIS
LIN {X -128.9718,Y 13.734,Z 147,A 170.2075,B 24.0811,C -1.3422,E1 23.9571,E2 276.5273} C_DIS
LIN {X -128.4658,Y 17.8633,Z 147,A 168.3229,B 24.0809,C -1.3461,E1 23.9577,E2 278.414} C_DIS
LIN {X -127.9184,Y 21.4293,Z 147,A 166.7695,B 24.0805,C -1.3531,E1 23.9584,E2 279.9597} C_DIS
LIN {X -127.157,Y 25.5634,Z 147,A 164.8929,B 24.0803,C -1.3582,E1 23.9594,E2 281.8353} C_DIS
LIN {X -126.5563,Y 28.3911,Z 147,A 163.5728,B 24.0801,C -1.3604,E1 23.9602,E2 283.158} C_DIS
LIN {X -125.7121,Y 31.9179,Z 147,A 162.0379,B 24.0797,C -1.3686,E1 23.9612,E2 284.6821} C_DIS
LIN {X -124.8839,Y 35.0185,Z 147,A 160.3133,B 24.0802,C -1.3595,E1 23.9625,E2 286.4396} C_DIS
LIN {X -123.5237,Y 39.5495,Z 147,A 158.4753,B 24.0792,C -1.3773,E1 23.964,E2 288.2447} C_DIS
LIN {X -122.1765,Y 43.5362,Z 147,A 156.5557,B 24.0791,C -1.3804,E1 23.9658,E2 290.168} C_DIS
LIN {X -121.129,Y 46.3731,Z 147,A 155.0946,B 24.0791,C -1.379,E1 23.9673,E2 291.6412} C_DIS
LIN {X -119.5582,Y 50.281,Z 147,A 153.348,B 24.0786,C -1.3898,E1 23.9691,E2 293.3712} C_DIS
LIN {X -117.8982,Y 54.0595,Z 147,A 151.6442,B 24.078,C -1.4007,E1 23.971,E2 295.0578} C_DIS
LIN {X -116.9218,Y 56.1389,Z 147,A 150.1605,B 24.0789,C -1.3829,E1 23.9729,E2 296.5938} C_DIS
LIN {X -115.2355,Y 59.5281,Z 147,A 148.7358,B 24.0781,C -1.3989,E1 23.9746,E2 297.987} C_DIS
LIN {X -113.1057,Y 63.4809,Z 147,A 146.8071,B 24.0776,C -1.4072,E1 23.9772,E2 299.9059} C_DIS
LIN {X -109.9182,Y 68.8539,Z 147,A 143.9714,B 24.0774,C -1.4118,E1 23.9813,E2 302.7455} C_DIS
LIN {X -107.5998,Y 72.4233,Z 147,A 142.0716,B 24.0771,C -1.4162,E1 23.9842,E2 304.6442} C_DIS
LIN {X -105.537,Y 75.3967,Z 147,A 140.4513,B 24.0769,C -1.4197,E1 23.9869,E2 306.2643} C_DIS
LIN {X -102.8079,Y 79.0784,Z 147,A 138.5448,B 24.0763,C -1.4305,E1 23.99,E2 308.1537} C_DIS
LIN {X -100.051,Y 82.5384,Z 147,A 136.5067,B 24.0763,C -1.4319,E1 23.9936,E2 310.1981} C_DIS
LIN {X -97.2778,Y 85.7891,Z 147,A 134.6662,B 24.0758,C -1.4389,E1 23.997,E2 312.0301} C_DIS
LIN {X -94.8006,Y 88.5189,Z 147,A 133.0262,B 24.0756,C -1.4425,E1 24.0001,E2 313.6687} C_DIS
LIN {X -92.2147,Y 91.21,Z 147,A 131.2705,B 24.0756,C -1.4418,E1 24.0035,E2 315.4342} C_DIS
LIN {X -89.069,Y 94.2838,Z 147,A 129.3922,B 24.0753,C -1.4494,E1 24.0073,E2 317.3019} C_DIS
LIN {X -86.1949,Y 96.9191,Z 147,A 127.6484,B 24.0751,C -1.4524,E1 24.0109,E2 319.0455} C_DIS
LIN {X -83.2484,Y 99.4607,Z 147,A 125.896,B 24.0749,C -1.4548,E1 24.0146,E2 320.7991} C_DIS
LIN {X -80.3861,Y 101.7886,Z 147,A 124.2266,B 24.0749,C -1.4565,E1 24.0183,E2 322.4708} C_DIS
LIN {X -77.2337,Y 104.2005,Z 147,A 122.5596,B 24.0744,C -1.4642,E1 24.0219,E2 324.1252} C_DIS
LIN {X -73.889,Y 106.5982,Z 147,A 120.8355,B 24.074,C -1.4722,E1 24.0258,E2 325.8358} C_DIS
LIN {X -70.9606,Y 108.5701,Z 147,A 119.054,B 24.0744,C -1.4651,E1 24.03,E2 327.6408} C_DIS
LIN {X -67.8421,Y 110.5449,Z 147,A 117.2223,B 24.0747,C -1.459,E1 24.0345,E2 329.4935} C_DIS
LIN {X -64.9532,Y 112.2667,Z 147,A 115.1564,B 24.076,C -1.4353,E1 24.0396,E2 331.6239} C_DIS
LIN {X -59.4698,Y 115.2652,Z 147,A 113.2249,B 24.0736,C -1.4777,E1 24.0441,E2 333.4567} C_DIS
LIN {X -56.1001,Y 116.9404,Z 147,A 111.6356,B 24.0733,C -1.4838,E1 24.0481,E2 335.0354} C_DIS
LIN {X -53.6215,Y 118.0995,Z 147,A 110.4235,B 24.0732,C -1.4854,E1 24.0512,E2 336.2466} C_DIS
LIN {X -50.5515,Y 119.4452,Z 147,A 108.843,B 24.0733,C -1.483,E1 24.0552,E2 337.8369} C_DIS
LIN {X -47.0473,Y 120.8669,Z 147,A 107.4841,B 24.0724,C -1.4998,E1 24.0587,E2 339.1578} C_DIS
LIN {X -43.2183,Y 122.2908,Z 147,A 105.387,B 24.073,C -1.4885,E1 24.0643,E2 341.287} C_DIS
LIN {X -38.3192,Y 123.9114,Z 147,A 103.1543,B 24.0727,C -1.4934,E1 24.0702,E2 343.5119} C_DIS
LIN {X -34.9271,Y 124.9094,Z 147,A 101.5796,B 24.0727,C -1.4945,E1 24.0744,E2 345.0866} C_DIS
LIN {X -31.3188,Y 125.8641,Z 147,A 99.815,B 24.0729,C -1.4907,E1 24.0792,E2 346.8631} C_DIS
LIN {X -27.5602,Y 126.739,Z 147,A 98.2233,B 24.0725,C -1.4976,E1 24.0835,E2 348.4401} C_DIS
LIN {X -24.7121,Y 127.3254,Z 147,A 96.8946,B 24.0725,C -1.4965,E1 24.0871,E2 349.7729} C_DIS
LIN {X -16.0329,Y 128.7079,Z 147,A 92.9319,B 24.0726,C -1.4953,E1 24.0981,E2 353.7421} C_DIS
LIN {X -12.9271,Y 129.0563,Z 147,A 90.8829,B 24.0744,C -1.4647,E1 24.104,E2 355.8673} C_DIS
LIN {X -7.2381,Y 129.501,Z 147,A 89.0707,B 24.0724,C -1.4989,E1 24.1088,E2 357.5963} C_DIS
LIN {X -0.863,Y 129.6983,Z 147,A 86.303,B 24.0722,C -1.502,E1 24.1165,E2 360.3566} C_DIS
LIN {X 2.982,Y 129.6683,Z 147,A 84.5498,B 24.0724,C -1.4997,E1 24.1214,E2 362.1155} C_DIS
LIN {X 7.3435,Y 129.4943,Z 147,A 82.1786,B 24.0736,C -1.4786,E1 24.1282,E2 364.5372} C_DIS
LIN {X 11.687,Y 129.1753,Z 147,A 80.6649,B 24.0725,C -1.498,E1 24.1323,E2 366.0028} C_DIS
LIN {X 14.6335,Y 128.8749,Z 147,A 79.0828,B 24.0732,C -1.4846,E1 24.1368,E2 367.6163} C_DIS
LIN {X 18.1039,Y 128.4314,Z 147,A 78.0812,B 24.0717,C -1.5104,E1 24.1394,E2 368.5541} C_DIS
LIN {X 23.0538,Y 127.6357,Z 147,A 75.6682,B 24.0723,C -1.5,E1 24.1461,E2 370.9898} C_DIS
LIN {X 27.1401,Y 126.8297,Z 147,A 73.9632,B 24.072,C -1.5057,E1 24.1507,E2 372.6788} C_DIS
LIN {X 29.6625,Y 126.2655,Z 147,A 72.7682,B 24.0722,C -1.5024,E1 24.1539,E2 373.88} C_DIS
LIN {X 33.3095,Y 125.3506,Z 147,A 71.0715,B 24.0724,C -1.4997,E1 24.1586,E2 375.5807} C_DIS
LIN {X 36.458,Y 124.4712,Z 147,A 69.6616,B 24.0724,C -1.5003,E1 24.1623,E2 376.9866} C_DIS
LIN {X 40.217,Y 123.3104,Z 147,A 67.7414,B 24.0729,C -1.49,E1 24.1675,E2 378.9283} C_DIS
LIN {X 43.8372,Y 122.0679,Z 147,A 66.2057,B 24.0726,C -1.4961,E1 24.1715,E2 380.446} C_DIS
LIN {X 46.6416,Y 121.0246,Z 147,A 64.8178,B 24.0728,C -1.4915,E1 24.1751,E2 381.8418} C_DIS
LIN {X 49.8704,Y 119.7297,Z 147,A 63.2395,B 24.073,C -1.4879,E1 24.1792,E2 383.4254} C_DIS
LIN {X 54.0667,Y 117.8948,Z 147,A 61.3082,B 24.073,C -1.49,E1 24.1841,E2 385.3464} C_DIS
LIN {X 57.4137,Y 116.3009,Z 147,A 59.7214,B 24.0729,C -1.4905,E1 24.1881,E2 386.9277} C_DIS
LIN {X 60.0215,Y 114.9771,Z 147,A 58.3709,B 24.0732,C -1.4859,E1 24.1915,E2 388.2856} C_DIS
LIN {X 63.4619,Y 113.1164,Z 147,A 56.5904,B 24.0735,C -1.4808,E1 24.1958,E2 390.073} C_DIS
LIN {X 67.4395,Y 110.7915,Z 147,A 54.5248,B 24.0737,C -1.4762,E1 24.2008,E2 392.1432} C_DIS
LIN {X 71.1011,Y 108.4778,Z 147,A 52.6382,B 24.0738,C -1.4745,E1 24.2052,E2 394.0277} C_DIS
LIN {X 74.8656,Y 105.9145,Z 147,A 50.6904,B 24.0738,C -1.4743,E1 24.2097,E2 395.9691} C_DIS
LIN {X 78.3369,Y 103.3737,Z 147,A 48.7602,B 24.0741,C -1.4694,E1 24.214,E2 397.904} C_DIS
LIN {X 81.8016,Y 100.6546,Z 147,A 46.789,B 24.0744,C -1.4644,E1 24.2183,E2 399.8797} C_DIS
LIN {X 85.2391,Y 97.76,Z 147,A 45.0994,B 24.0738,C -1.4753,E1 24.2219,E2 401.5358} C_DIS
LIN {X 87.5282,Y 95.7165,Z 147,A 43.6555,B 24.0742,C -1.4681,E1 24.2249,E2 402.9913} C_DIS
LIN {X 91.4521,Y 91.9741,Z 147,A 40.2346,B 24.0774,C -1.4118,E1 24.2319,E2 406.5346} C_DIS
LIN {X 96.053,Y 87.1581,Z 147,A 38.2023,B 24.0752,C -1.4505,E1 24.2356,E2 408.4632} C_DIS
LIN {X 99.0149,Y 83.7787,Z 147,A 36.2053,B 24.0755,C -1.4453,E1 24.2392,E2 410.4636} C_DIS
LIN {X 101.7384,Y 80.4499,Z 147,A 34.294,B 24.0758,C -1.4401,E1 24.2426,E2 412.3782} C_DIS
LIN {X 104.4101,Y 76.9499,Z 147,A 32.4025,B 24.0759,C -1.4379,E1 24.2457,E2 414.2655} C_DIS
LIN {X 106.8744,Y 73.4888,Z 147,A 30.5189,B 24.0762,C -1.4328,E1 24.2488,E2 416.1521} C_DIS
LIN {X 109.3597,Y 69.7369,Z 147,A 28.549,B 24.0764,C -1.4285,E1 24.2518,E2 418.1223} C_DIS
LIN {X 111.4685,Y 66.3137,Z 147,A 26.8184,B 24.0766,C -1.426,E1 24.2543,E2 419.8497} C_DIS
LIN {X 113.664,Y 62.477,Z 147,A 24.8245,B 24.077,C -1.4185,E1 24.257,E2 421.851} C_DIS
LIN {X 115.4528,Y 59.1012,Z 147,A 23.2992,B 24.0768,C -1.4221,E1 24.259,E2 423.359} C_DIS
LIN {X 116.6205,Y 56.7658,Z 147,A 22.1276,B 24.077,C -1.4179,E1 24.2604,E2 424.5345} C_DIS
LIN {X 118.2272,Y 53.336,Z 147,A 20.3803,B 24.0775,C -1.4093,E1 24.2625,E2 426.293} C_DIS
LIN {X 120.7294,Y 47.401,Z 147,A 17.5953,B 24.0778,C -1.404,E1 24.2654,E2 429.0749} C_DIS
LIN {X 122.1003,Y 43.7473,Z 147,A 15.8785,B 24.078,C -1.3992,E1 24.2671,E2 430.7934} C_DIS
LIN {X 123.4378,Y 39.8185,Z 147,A 14.0722,B 24.0783,C -1.395,E1 24.2687,E2 432.5992} C_DIS
LIN {X 124.4455,Y 36.5459,Z 147,A 12.6448,B 24.0783,C -1.3947,E1 24.2698,E2 434.0188} C_DIS
LIN {X 125.3194,Y 33.4263,Z 147,A 11.1914,B 24.0786,C -1.3892,E1 24.2709,E2 435.4771} C_DIS
LIN {X 126.0967,Y 30.363,Z 147,A 9.8282,B 24.0787,C -1.3865,E1 24.2718,E2 436.8386} C_DIS
LIN {X 126.6607,Y 27.923,Z 147,A 8.7883,B 24.0787,C -1.3865,E1 24.2724,E2 437.8724} C_DIS
LIN {X 127.3612,Y 24.5249,Z 147,A 7.1332,B 24.0793,C -1.3753,E1 24.2734,E2 439.5446} C_DIS
LIN {X 128.3753,Y 18.4967,Z 147,A 4.2425,B 24.0803,C -1.3568,E1 24.2746,E2 442.4626} C_DIS
LIN {X 128.9065,Y 14.3412,Z 147,A 2.1498,B 24.0813,C -1.3384,E1 24.2753,E2 444.5873} C_DIS
LIN {X 129.3069,Y 10.1266,Z 147,A 0.6635,B 24.0806,C -1.352,E1 24.2757,E2 446.0311} C_DIS
LIN {X 129.5556,Y 6.1514,Z 147,A -1.0426,B 24.0807,C -1.3491,E1 24.2759,E2 447.7338} C_DIS
LIN {X 129.6766,Y 2.549,Z 147,A -2.6314,B 24.081,C -1.3441,E1 24.276,E2 449.3251} C_DIS
LIN {X 129.6719,Y -2.8302,Z 147,A -5.0193,B 24.0814,C -1.3357,E1 24.276,E2 451.7186} C_DIS
LIN {X 129.5183,Y -6.8929,Z 147,A -6.9331,B 24.0821,C -1.3237,E1 24.2757,E2 453.6497} C_DIS
LIN {X 129.1479,Y -11.9727,Z 147,A -8.7781,B 24.0814,C -1.3373,E1 24.2753,E2 455.4502} C_DIS
LIN {X 128.6665,Y -16.3557,Z 147,A -10.9253,B 24.0822,C -1.3206,E1 24.2746,E2 457.6249} C_DIS
LIN {X 128.1612,Y -19.9254,Z 147,A -12.4542,B 24.0823,C -1.3187,E1 24.274,E2 459.149} C_DIS
LIN {X 127.5875,Y -23.323,Z 147,A -14.3945,B 24.0837,C -1.2921,E1 24.273,E2 461.1422} C_DIS
LIN {X 126.8286,Y -27.145,Z 147,A -15.6281,B 24.0827,C -1.3117,E1 24.2723,E2 462.3205} C_DIS
LIN {X 126.1256,Y -30.2432,Z 147,A -17.0128,B 24.0829,C -1.3082,E1 24.2715,E2 463.7055} C_DIS
LIN {X 125.4122,Y -33.0785,Z 147,A -18.2397,B 24.0829,C -1.3074,E1 24.2706,E2 464.9271} C_DIS
LIN {X 124.7174,Y -35.614,Z 147,A -19.6497,B 24.0837,C -1.2907,E1 24.2695,E2 466.3692} C_DIS
LIN {X 123.6632,Y -39.1128,Z 147,A -21.1346,B 24.0837,C -1.2923,E1 24.2683,E2 467.8415} C_DIS
LIN {X 122.5397,Y -42.5003,Z 147,A -22.6223,B 24.0837,C -1.2919,E1 24.267,E2 469.3214} C_DIS
LIN {X 121.4676,Y -45.4738,Z 147,A -24.0257,B 24.0839,C -1.2871,E1 24.2656,E2 470.7282} C_DIS
LIN {X 120.5206,Y -47.9311,Z 147,A -25.5127,B 24.0849,C -1.2668,E1 24.2641,E2 472.2563} C_DIS
LIN {X 119.277,Y -50.9467,Z 147,A -26.6416,B 24.0844,C -1.2784,E1 24.2629,E2 473.3504} C_DIS
LIN {X 118.2806,Y -53.2166,Z 147,A -28.6613,B 24.0869,C -1.2276,E1 24.2604,E2 475.4824} C_DIS
LIN {X 115.4767,Y -59.0542,Z 147,A -30.5801,B 24.0849,C -1.2672,E1 24.2581,E2 477.2941} C_DIS
LIN {X 113.6779,Y -62.4518,Z 147,A -32.3726,B 24.0854,C -1.2572,E1 24.2557,E2 479.1011} C_DIS
LIN {X 111.9912,Y -65.4278,Z 147,A -33.8949,B 24.0857,C -1.2522,E1 24.2536,E2 480.6274} C_DIS
LIN {X 109.5425,Y -69.4495,Z 147,A -35.8729,B 24.0857,C -1.2514,E1 24.2507,E2 482.5969} C_DIS
LIN {X 107.1776,Y -73.0469,Z 147,A -37.803,B 24.086,C -1.2446,E1 24.2477,E2 484.5338} C_DIS
LIN {X 104.7315,Y -76.5125,Z 147,A -39.6298,B 24.0862,C -1.2418,E1 24.2447,E2 486.3581} C_DIS
LIN {X 100.1939,Y -82.3654,Z 147,A -42.9525,B 24.0867,C -1.2303,E1 24.239,E2 489.6926} C_DIS
LIN {X 97.3505,Y -85.7069,Z 147,A -44.7003,B 24.0865,C -1.235,E1 24.2358,E2 491.4207} C_DIS
LIN {X 94.8851,Y -88.4282,Z 147,A -46.6513,B 24.0875,C -1.214,E1 24.232,E2 493.414} C_DIS
LIN {X 90.2741,Y -93.1306,Z 147,A -49.3517,B 24.0873,C -1.2175,E1 24.2267,E2 496.0939} C_DIS
LIN {X 86.9583,Y -96.2344,Z 147,A -51.2556,B 24.0873,C -1.2179,E1 24.2228,E2 497.9887} C_DIS
LIN {X 84.4868,Y -98.4111,Z 147,A -52.8179,B 24.0877,C -1.2091,E1 24.2195,E2 499.5662} C_DIS
LIN {X 80.1989,Y -101.9356,Z 147,A -55.2382,B 24.0879,C -1.2052,E1 24.2143,E2 501.9864} C_DIS
LIN {X 76.6552,Y -104.6266,Z 147,A -57.1638,B 24.088,C -1.2031,E1 24.21,E2 503.9101} C_DIS
LIN {X 73.3741,Y -106.9531,Z 147,A -59.3723,B 24.0892,C -1.1776,E1 24.2048,E2 506.1727} C_DIS
LIN {X 69.8197,Y -109.3067,Z 147,A -60.6002,B 24.0878,C -1.207,E1 24.2021,E2 507.3248} C_DIS
LIN {X 67.6817,Y -110.643,Z 147,A -62.881,B 24.0906,C -1.1463,E1 24.1963,E2 509.7464} C_DIS
LIN {X 61.6639,Y -114.1069,Z 147,A -65.0097,B 24.0887,C -1.1877,E1 24.1914,E2 511.7675} C_DIS
LIN {X 57.8941,Y -116.0639,Z 147,A -66.8134,B 24.0887,C -1.1882,E1 24.1869,E2 513.5648} C_DIS
LIN {X 55.2752,Y -117.3345,Z 147,A -68.2427,B 24.0891,C -1.1789,E1 24.1832,E2 515.0129} C_DIS
LIN {X 49.2801,Y -119.9761,Z 147,A -70.9881,B 24.089,C -1.182,E1 24.1762,E2 517.7439} C_DIS
LIN {X 45.7003,Y -121.3828,Z 147,A -72.6388,B 24.089,C -1.1821,E1 24.1719,E2 519.3906} C_DIS
LIN {X 42.6632,Y -122.4832,Z 147,A -74.0785,B 24.0891,C -1.1796,E1 24.1681,E2 520.8334} C_DIS
LIN {X 37.4379,Y -124.1812,Z 147,A -76.6059,B 24.0895,C -1.1717,E1 24.1614,E2 523.3753} C_DIS
LIN {X 33.5163,Y -125.2955,Z 147,A -78.2947,B 24.0893,C -1.1753,E1 24.1568,E2 525.0523} C_DIS
LIN {X 30.1724,Y -126.1426,Z 147,A -79.9077,B 24.0896,C -1.1694,E1 24.1524,E2 526.6774} C_DIS
LIN {X 26.4591,Y -126.9748,Z 147,A -81.5723,B 24.0896,C -1.1686,E1 24.1479,E2 528.3416} C_DIS
LIN {X 23.5082,Y -127.5544,Z 147,A -83.1105,B 24.0901,C -1.1572,E1 24.1436,E2 529.906} C_DIS
LIN {X 18.0315,Y -128.4418,Z 147,A -85.3012,B 24.0896,C -1.1683,E1 24.1376,E2 532.0675} C_DIS
LIN {X 12.5263,Y -129.0947,Z 147,A -87.6886,B 24.0896,C -1.1699,E1 24.131,E2 534.4492} C_DIS
LIN {X 8.8657,Y -129.3989,Z 147,A -89.4074,B 24.0898,C -1.1644,E1 24.1262,E2 536.1806} C_DIS
LIN {X 4.0203,Y -129.6394,Z 147,A -91.4449,B 24.0896,C -1.1687,E1 24.1205,E2 538.2067} C_DIS
LIN {X 0.9268,Y -129.6924,Z 147,A -92.7958,B 24.0896,C -1.1692,E1 24.1168,E2 539.5562} C_DIS
Enddeposition()
LIN {X 0.9268,Y -129.6924,Z 147,A -92.7958,B 24.0896,C -1.1692,E1 24.1168,E2 539.5562} C_DIS
Startdeposition()
$VEL.CP = VEL_PRINT
LIN {X 3.3366,Y -128.7036,Z 147,A -90.9809,B 23.2453,C -1.0564,E1 23.2731,E2 537.9146} C_DIS
LIN {X 9.7851,Y -128.3748,Z 147,A -87.896,B 23.2448,C -1.0675,E1 23.2817,E2 534.8028} C_DIS
LIN {X 15.14,Y -127.8532,Z 147,A -85.4871,B 23.2448,C -1.0695,E1 23.2884,E2 532.3906} C_DIS
LIN {X 18.1489,Y -127.4608,Z 147,A -83.5823,B 23.2435,C -1.0971,E1 23.2939,E2 530.4178} C_DIS
LIN {X 23.0121,Y -126.6735,Z 147,A -81.9201,B 23.2446,C -1.0732,E1 23.2983,E2 528.818} C_DIS
LIN {X 26.8864,Y -125.908,Z 147,A -80.2898,B 23.2448,C -1.0686,E1 23.3027,E2 527.2015} C_DIS
LIN {X 29.9133,Y -125.2233,Z 147,A -78.8962,B 23.2447,C -1.0705,E1 23.3065,E2 525.8051} C_DIS
LIN {X 33.1469,Y -124.4061,Z 147,A -77.4254,B 23.2447,C -1.0714,E1 23.3105,E2 524.3346} C_DIS
LIN {X 36.3178,Y -123.5177,Z 147,A -75.9851,B 23.2447,C -1.0718,E1 23.3143,E2 522.8959} C_DIS
LIN {X 45.2167,Y -120.5447,Z 147,A -72.1357,B 23.2451,C -1.0611,E1 23.3245,E2 519.0816} C_DIS
LIN {X 53.1796,Y -117.2515,Z 147,A -67.8172,B 23.2438,C -1.09,E1 23.3357,E2 514.7012} C_DIS
LIN {X 56.8397,Y -115.5197,Z 147,A -66.2823,B 23.2443,C -1.0799,E1 23.3395,E2 513.1962} C_DIS
LIN {X 61.2074,Y -113.2686,Z 147,A -64.1718,B 23.2443,C -1.0799,E1 23.3447,E2 511.0923} C_DIS
LIN {X 65.5205,Y -110.8287,Z 147,A -61.4689,B 23.243,C -1.1082,E1 23.3514,E2 508.3266} C_DIS
LIN {X 68.4357,Y -109.0536,Z 147,A -60.1872,B 23.2434,C -1.0994,E1 23.3544,E2 507.0715} C_DIS
LIN {X 73.9649,Y -105.3818,Z 147,A -56.3958,B 23.2413,C -1.1469,E1 23.3633,E2 503.1742} C_DIS
LIN {X 79.1912,Y -101.5133,Z 147,A -54.5685,B 23.2434,C -1.1001,E1 23.3671,E2 501.4723} C_DIS
LIN {X 83.7549,Y -97.7818,Z 147,A -52.0074,B 23.2433,C -1.1028,E1 23.3726,E2 498.915} C_DIS
LIN {X 87.8572,Y -94.1126,Z 147,A -49.3797,B 23.2426,C -1.1173,E1 23.3781,E2 496.2622} C_DIS
LIN {X 93.5474,Y -88.4586,Z 147,A -46.1413,B 23.243,C -1.1095,E1 23.3844,E2 493.0582} C_DIS
LIN {X 97.6074,Y -83.9573,Z 147,A -43.1644,B 23.242,C -1.1302,E1 23.39,E2 490.0435} C_DIS
LIN {X 100.4841,Y -80.4915,Z 147,A -40.8176,B 23.241,C -1.1526,E1 23.3942,E2 487.652} C_DIS
LIN {X 102.7043,Y -77.6394,Z 147,A -39.512,B 23.2415,C -1.1418,E1 23.3964,E2 486.3804} C_DIS
LIN {X 105.1889,Y -74.2383,Z 147,A -37.6394,B 23.2413,C -1.1469,E1 23.3994,E2 484.5048} C_DIS
LIN {X 107.0478,Y -71.5318,Z 147,A -35.8406,B 23.2403,C -1.168,E1 23.4023,E2 482.6627} C_DIS
LIN {X 109.1765,Y -68.2393,Z 147,A -34.7092,B 23.2415,C -1.1422,E1 23.4039,E2 481.6025} C_DIS
LIN {X 111.6082,Y -64.1855,Z 147,A -32.3319,B 23.2405,C -1.1619,E1 23.4073,E2 479.1886} C_DIS
LIN {X 113.7198,Y -60.3628,Z 147,A -30.626,B 23.2408,C -1.1558,E1 23.4096,E2 477.5079} C_DIS
LIN {X 115.4472,Y -56.9866,Z 147,A -28.5288,B 23.2396,C -1.1814,E1 23.4122,E2 475.3583} C_DIS
LIN {X 116.8713,Y -54.006,Z 147,A -27.4965,B 23.2405,C -1.1638,E1 23.4134,E2 474.3762} C_DIS
LIN {X 118.1669,Y -51.1091,Z 147,A -26.0164,B 23.2401,C -1.1715,E1 23.4151,E2 472.8855} C_DIS
LIN {X 119.2395,Y -48.5562,Z 147,A -24.8426,B 23.2401,C -1.1724,E1 23.4163,E2 471.7166} C_DIS
LIN {X 120.5192,Y -45.2847,Z 147,A -23.2474,B 23.2397,C -1.1788,E1 23.4179,E2 470.1147} C_DIS
LIN {X 121.5952,Y -42.3107,Z 147,A -21.8104,B 23.2395,C -1.1847,E1 23.4193,E2 468.6717} C_DIS
LIN {X 122.6244,Y -39.2279,Z 147,A -20.4126,B 23.2394,C -1.1868,E1 23.4205,E2 467.2771} C_DIS
LIN {X 123.436,Y -36.5969,Z 147,A -19.0596,B 23.2389,C -1.1971,E1 23.4216,E2 465.9065} C_DIS
LIN {X 124.5261,Y -32.6969,Z 147,A -17.2312,B 23.2385,C -1.2042,E1 23.4229,E2 464.0718} C_DIS
LIN {X 125.4741,Y -28.8426,Z 147,A -15.5504,B 23.2385,C -1.2055,E1 23.424,E2 462.3981} C_DIS
LIN {X 126.1639,Y -25.6568,Z 147,A -13.1588,B 23.2358,C -1.2579,E1 23.4254,E2 459.8896} C_DIS
LIN {X 127.3595,Y -18.8576,Z 147,A -11.2005,B 23.2382,C -1.2113,E1 23.4262,E2 458.0613} C_DIS
LIN {X 127.707,Y -16.3316,Z 147,A -9.3095,B 23.2361,C -1.2532,E1 23.4269,E2 456.0768} C_DIS
LIN {X 128.2599,Y -11.188,Z 147,A -7.9054,B 23.238,C -1.2153,E1 23.4272,E2 454.7773} C_DIS
LIN {X 128.6694,Y -4.4877,Z 147,A -4.8304,B 23.2373,C -1.2293,E1 23.4277,E2 451.6867} C_DIS
LIN {X 128.7368,Y 1.6576,Z 147,A -2.0568,B 23.2367,C -1.2401,E1 23.4277,E2 448.9039} C_DIS
LIN {X 128.5593,Y 6.9593,Z 147,A 0.4243,B 23.236,C -1.2537,E1 23.4274,E2 446.4044} C_DIS
LIN {X 128.1269,Y 12.6191,Z 147,A 3.1287,B 23.2352,C -1.2708,E1 23.4268,E2 443.6743} C_DIS
LIN {X 127.7545,Y 15.9675,Z 147,A 5.0389,B 23.2338,C -1.2964,E1 23.4261,E2 441.712} C_DIS
LIN {X 126.9901,Y 21.1927,Z 147,A 6.7234,B 23.2352,C -1.2702,E1 23.4254,E2 440.1041} C_DIS
LIN {X 126.1853,Y 25.5518,Z 147,A 8.6128,B 23.2351,C -1.2723,E1 23.4244,E2 438.2215} C_DIS
LIN {X 125.3852,Y 29.2317,Z 147,A 10.3979,B 23.2345,C -1.2829,E1 23.4233,E2 436.4208} C_DIS
LIN {X 124.5029,Y 32.784,Z 147,A 11.871,B 23.2347,C -1.2802,E1 23.4222,E2 434.9639} C_DIS
LIN {X 123.6899,Y 35.7297,Z 147,A 13.2888,B 23.2343,C -1.2872,E1 23.4212,E2 433.537} C_DIS
LIN {X 122.662,Y 39.1104,Z 147,A 14.7896,B 23.2343,C -1.2884,E1 23.4199,E2 432.0424} C_DIS
LIN {X 121.6314,Y 42.2062,Z 147,A 16.255,B 23.234,C -1.2935,E1 23.4186,E2 430.5733} C_DIS
LIN {X 120.1982,Y 46.1331,Z 147,A 17.9715,B 23.234,C -1.2918,E1 23.4169,E2 428.8714} C_DIS
LIN {X 118.9024,Y 49.3746,Z 147,A 19.8293,B 23.233,C -1.3115,E1 23.4149,E2 426.9751} C_DIS
LIN {X 116.8872,Y 53.9716,Z 147,A 21.8376,B 23.2333,C -1.3067,E1 23.4127,E2 424.9906} C_DIS
LIN {X 115.7031,Y 56.4679,Z 147,A 23.1418,B 23.2329,C -1.3139,E1 23.4111,E2 423.676} C_DIS
LIN {X 114.0765,Y 59.6834,Z 147,A 24.63,B 23.2329,C -1.3127,E1 23.4092,E2 422.1994} C_DIS
LIN {X 112.7606,Y 62.1382,Z 147,A 26.0174,B 23.2324,C -1.3234,E1 23.4073,E2 420.793} C_DIS
LIN {X 110.4348,Y 66.1838,Z 147,A 27.8466,B 23.2327,C -1.3167,E1 23.4047,E2 418.9906} C_DIS
LIN {X 108.4725,Y 69.3524,Z 147,A 29.6805,B 23.232,C -1.3298,E1 23.402,E2 417.1339} C_DIS
LIN {X 106.0869,Y 72.9494,Z 147,A 31.6002,B 23.2318,C -1.3347,E1 23.399,E2 415.2122} C_DIS
LIN {X 103.5167,Y 76.5539,Z 147,A 33.613,B 23.2314,C -1.3417,E1 23.3957,E2 413.1922} C_DIS
LIN {X 100.8246,Y 80.0652,Z 147,A 35.5363,B 23.2313,C -1.3443,E1 23.3924,E2 411.2723} C_DIS
LIN {X 98.0251,Y 83.4693,Z 147,A 37.4729,B 23.2311,C -1.3477,E1 23.3889,E2 409.3367} C_DIS
LIN {X 95.0661,Y 86.8253,Z 147,A 39.6242,B 23.2304,C -1.3601,E1 23.3848,E2 407.1645} C_DIS
LIN {X 90.9955,Y 91.0823,Z 147,A 41.7834,B 23.2313,C -1.3432,E1 23.3808,E2 405.0578} C_DIS
LIN {X 88.6822,Y 93.3354,Z 147,A 43.4802,B 23.2305,C -1.3589,E1 23.3773,E2 403.3291} C_DIS
LIN {X 85.5354,Y 96.2281,Z 147,A 45.4291,B 23.2301,C -1.3651,E1 23.3732,E2 401.3732} C_DIS
LIN {X 82.2119,Y 99.0821,Z 147,A 47.3342,B 23.2301,C -1.3667,E1 23.3692,E2 399.472} C_DIS
LIN {X 78.6462,Y 101.9357,Z 147,A 49.3734,B 23.2298,C -1.3708,E1 23.3647,E2 397.4306} C_DIS
LIN {X 75.1176,Y 104.5632,Z 147,A 51.2961,B 23.2297,C -1.3725,E1 23.3603,E2 395.5108} C_DIS
LIN {X 71.8864,Y 106.8106,Z 147,A 53.0933,B 23.2294,C -1.3777,E1 23.3562,E2 393.7073} C_DIS
LIN {X 68.4449,Y 109.0479,Z 147,A 54.6063,B 23.2301,C -1.3655,E1 23.3527,E2 392.2304} C_DIS
LIN {X 65.585,Y 110.7916,Z 147,A 56.2081,B 23.2297,C -1.3731,E1 23.3489,E2 390.6149} C_DIS
LIN {X 61.9385,Y 112.8706,Z 147,A 58.1926,B 23.2292,C -1.3813,E1 23.344,E2 388.6159} C_DIS
LIN {X 58.9425,Y 114.4625,Z 147,A 59.7252,B 23.229,C -1.3844,E1 23.3402,E2 387.0801} C_DIS
LIN {X 55.6864,Y 116.0802,Z 147,A 61.2451,B 23.2292,C -1.3818,E1 23.3364,E2 385.5712} C_DIS
LIN {X 52.7639,Y 117.4375,Z 147,A 62.7469,B 23.2289,C -1.3867,E1 23.3326,E2 384.0611} C_DIS
LIN {X 47.7263,Y 119.574,Z 147,A 65.3549,B 23.2283,C -1.3975,E1 23.3258,E2 381.4323} C_DIS
LIN {X 43.5005,Y 121.1747,Z 147,A 67.1285,B 23.2288,C -1.3882,E1 23.3212,E2 379.6863} C_DIS
LIN {X 39.731,Y 122.4637,Z 147,A 69.1137,B 23.2282,C -1.3997,E1 23.3159,E2 377.6761} C_DIS
LIN {X 34.893,Y 123.9279,Z 147,A 71.1485,B 23.2286,C -1.3912,E1 23.3105,E2 375.6665} C_DIS
LIN {X 31.515,Y 124.8296,Z 147,A 72.6924,B 23.2286,C -1.3917,E1 23.3063,E2 374.1241} C_DIS
LIN {X 27.7699,Y 125.7172,Z 147,A 74.3774,B 23.2286,C -1.3913,E1 23.3017,E2 372.4426} C_DIS
LIN {X 24.3675,Y 126.4195,Z 147,A 75.9517,B 23.2286,C -1.3933,E1 23.2974,E2 370.8652} C_DIS
LIN {X 20.3806,Y 127.1249,Z 147,A 77.9246,B 23.228,C -1.4019,E1 23.2919,E2 368.8726} C_DIS
LIN {X 16.7806,Y 127.6482,Z 147,A 80.0064,B 23.2268,C -1.424,E1 23.286,E2 366.7367} C_DIS
LIN {X 11.805,Y 128.2051,Z 147,A 81.5493,B 23.2286,C -1.3923,E1 23.282,E2 365.2753} C_DIS
LIN {X 5.7217,Y 128.6213,Z 147,A 84.242,B 23.2286,C -1.3914,E1 23.2745,E2 362.5862} C_DIS
LIN {X -0.6669,Y 128.7449,Z 147,A 86.9986,B 23.2289,C -1.3869,E1 23.2668,E2 359.8412} C_DIS
LIN {X -7.8189,Y 128.5089,Z 147,A 90.033,B 23.2293,C -1.379,E1 23.2584,E2 356.8263} C_DIS
LIN {X -14.0463,Y 127.9782,Z 147,A 93.2244,B 23.2284,C -1.3964,E1 23.2494,E2 353.5891} C_DIS
LIN {X -19.187,Y 127.3089,Z 147,A 95.9057,B 23.2275,C -1.4121,E1 23.2418,E2 350.8657} C_DIS
LIN {X -23.304,Y 126.6213,Z 147,A 97.3933,B 23.2285,C -1.3937,E1 23.2379,E2 349.423} C_DIS
LIN {X -27.0691,Y 125.8685,Z 147,A 99.0106,B 23.2288,C -1.3882,E1 23.2335,E2 347.8177} C_DIS
LIN {X -30.4805,Y 125.0865,Z 147,A 100.6489,B 23.2287,C -1.3904,E1 23.229,E2 346.1714} C_DIS
LIN {X -34.4256,Y 124.0586,Z 147,A 102.3987,B 23.229,C -1.3856,E1 23.2243,E2 344.4308} C_DIS
LIN {X -37.6408,Y 123.1209,Z 147,A 103.8275,B 23.2292,C -1.3812,E1 23.2205,E2 343.0105} C_DIS
LIN {X -40.9467,Y 122.0615,Z 147,A 105.4324,B 23.2292,C -1.3821,E1 23.2163,E2 341.4002} C_DIS
LIN {X -44.5942,Y 120.7778,Z 147,A 107.2666,B 23.229,C -1.385,E1 23.2114,E2 339.5547} C_DIS
LIN {X -48.3926,Y 119.3055,Z 147,A 108.9821,B 23.2294,C -1.3782,E1 23.207,E2 337.8525} C_DIS
LIN {X -51.186,Y 118.1336,Z 147,A 110.4342,B 23.2292,C -1.3809,E1 23.2032,E2 336.3898} C_DIS
LIN {X -55.131,Y 116.3455,Z 147,A 112.2827,B 23.2296,C -1.3744,E1 23.1986,E2 334.5528} C_DIS
LIN {X -59.0392,Y 114.4133,Z 147,A 114.7499,B 23.2284,C -1.3948,E1 23.1923,E2 332.0265} C_DIS
LIN {X -62.9535,Y 112.3072,Z 147,A 116.4703,B 23.2293,C -1.3799,E1 23.1882,E2 330.3388} C_DIS
LIN {X -66.7658,Y 110.0836,Z 147,A 118.2441,B 23.23,C -1.3678,E1 23.184,E2 328.5897} C_DIS
LIN {X -70.4474,Y 107.7653,Z 147,A 120.0847,B 23.2304,C -1.3599,E1 23.1797,E2 326.7629} C_DIS
LIN {X -73.981,Y 105.3704,Z 147,A 122.1304,B 23.2302,C -1.3626,E1 23.175,E2 324.7028} C_DIS
LIN {X -77.1653,Y 103.0615,Z 147,A 124.135,B 23.2298,C -1.3702,E1 23.1704,E2 322.6711} C_DIS
LIN {X -79.9436,Y 100.9215,Z 147,A 125.4504,B 23.2306,C -1.356,E1 23.1676,E2 321.3866} C_DIS
LIN {X -83.224,Y 98.2336,Z 147,A 127.3361,B 23.2308,C -1.3518,E1 23.1635,E2 319.5038} C_DIS
LIN {X -86.535,Y 95.3295,Z 147,A 129.2301,B 23.2312,C -1.3444,E1 23.1596,E2 317.6204} C_DIS
LIN {X -90.1436,Y 91.9248,Z 147,A 131.4758,B 23.2314,C -1.3408,E1 23.1551,E2 315.3738} C_DIS
LIN {X -93.1745,Y 88.8514,Z 147,A 133.4111,B 23.2317,C -1.3367,E1 23.1513,E2 313.4398} C_DIS
LIN {X -96.0936,Y 85.6862,Z 147,A 135.6316,B 23.2312,C -1.3452,E1 23.1471,E2 311.187} C_DIS
LIN {X -98.3535,Y 83.0829,Z 147,A 136.9383,B 23.232,C -1.3313,E1 23.1448,E2 309.9093} C_DIS
LIN {X -102.7847,Y 77.5328,Z 147,A 140.515,B 23.2314,C -1.3411,E1 23.1386,E2 306.2893} C_DIS
LIN {X -105.2738,Y 74.118,Z 147,A 141.9797,B 23.2327,C -1.3177,E1 23.1363,E2 304.8763} C_DIS
LIN {X -107.7622,Y 70.4522,Z 147,A 144.0169,B 23.2328,C -1.3151,E1 23.1332,E2 302.8349} C_DIS
LIN {X -113.1218,Y 61.4779,Z 147,A 148.2209,B 23.2346,C -1.2822,E1 23.1273,E2 298.6911} C_DIS
LIN {X -116.3058,Y 55.2142,Z 147,A 151.8206,B 23.234,C -1.2932,E1 23.1227,E2 295.0424} C_DIS
LIN {X -118.0722,Y 51.3281,Z 147,A 153.5248,B 23.2347,C -1.279,E1 23.1208,E2 293.3642} C_DIS
LIN {X -119.2547,Y 48.5186,Z 147,A 154.8633,B 23.235,C -1.2741,E1 23.1194,E2 292.0302} C_DIS
LIN {X -121.4268,Y 42.7966,Z 147,A 157.828,B 23.2349,C -1.2759,E1 23.1165,E2 289.0425} C_DIS
LIN {X -122.5715,Y 39.3937,Z 147,A 160.185,B 23.2334,C -1.3039,E1 23.1144,E2 286.5995} C_DIS
LIN {X -124.2515,Y 33.7266,Z 147,A 162.0876,B 23.2355,C -1.2639,E1 23.113,E2 284.787} C_DIS
LIN {X -125.1676,Y 30.1443,Z 147,A 163.6601,B 23.2359,C -1.2556,E1 23.112,E2 283.2259} C_DIS
LIN {X -125.9375,Y 26.7497,Z 147,A 165.3154,B 23.2359,C -1.2552,E1 23.111,E2 281.561} C_DIS
LIN {X -126.7149,Y 22.781,Z 147,A 167.0222,B 23.2365,C -1.2454,E1 23.1101,E2 279.8681} C_DIS
LIN {X -127.2707,Y 19.4389,Z 147,A 168.6116,B 23.2365,C -1.244,E1 23.1094,E2 278.2719} C_DIS
LIN {X -127.7928,Y 15.6464,Z 147,A 170.371,B 23.2367,C -1.2409,E1 23.1088,E2 276.5091} C_DIS
LIN {X -128.2558,Y 11.2365,Z 147,A 172.3154,B 23.2371,C -1.2333,E1 23.1083,E2 274.5715} C_DIS
LIN {X -128.5205,Y 7.6311,Z 147,A 173.9361,B 23.2373,C -1.2286,E1 23.108,E2 272.9522} C_DIS
LIN {X -128.701,Y 3.4305,Z 147,A 175.7671,B 23.2377,C -1.2208,E1 23.1078,E2 271.129} C_DIS
LIN {X -128.7483,Y -0.288,Z 147,A 177.4817,B 23.2378,C -1.218,E1 23.1078,E2 269.4105} C_DIS
LIN {X -128.6926,Y -3.7307,Z 147,A 178.9916,B 23.2381,C -1.2121,E1 23.1078,E2 267.9057} C_DIS
LIN {X -128.5087,Y -7.8225,Z 147,A -179.2207,B 23.2385,C -1.2047,E1 23.1081,E2 266.1251} C_DIS
LIN {X -128.2469,Y -11.3428,Z 147,A -177.4844,B 23.2384,C -1.2068,E1 23.1085,E2 264.3722} C_DIS
LIN {X -127.8402,Y -15.2487,Z 147,A -175.817,B 23.2388,C -1.1978,E1 23.109,E2 262.717} C_DIS
LIN {X -127.2709,Y -19.4379,Z 147,A -173.9378,B 23.2391,C -1.1917,E1 23.1098,E2 260.8411} C_DIS
LIN {X -126.7117,Y -22.7989,Z 147,A -172.4161,B 23.2393,C -1.1872,E1 23.1105,E2 259.3212} C_DIS
LIN {X -125.9273,Y -26.797,Z 147,A -170.5658,B 23.2395,C -1.1831,E1 23.1115,E2 257.4695} C_DIS
LIN {X -125.1126,Y -30.3724,Z 147,A -168.9322,B 23.2398,C -1.1781,E1 23.1126,E2 255.8381} C_DIS
LIN {X -123.5528,Y -36.1978,Z 147,A -166.236,B 23.2401,C -1.1704,E1 23.1146,E2 253.1446} C_DIS
LIN {X -122.3963,Y -39.9408,Z 147,A -164.2903,B 23.24,C -1.1739,E1 23.1163,E2 251.178} C_DIS
LIN {X -120.5217,Y -45.278,Z 147,A -161.8816,B 23.2406,C -1.1617,E1 23.1185,E2 248.7856} C_DIS
LIN {X -118.8901,Y -49.404,Z 147,A -160.0279,B 23.2411,C -1.1507,E1 23.1204,E2 246.9488} C_DIS
LIN {X -117.674,Y -52.2351,Z 147,A -158.5299,B 23.2411,C -1.1522,E1 23.1221,E2 245.4378} C_DIS
LIN {X -116.1724,Y -55.4934,Z 147,A -156.9858,B 23.2413,C -1.1454,E1 23.124,E2 243.9019} C_DIS
LIN {X -114.7376,Y -58.4023,Z 147,A -155.2443,B 23.2409,C -1.1544,E1 23.1262,E2 242.1273} C_DIS
LIN {X -113.2031,Y -61.3275,Z 147,A -154.0402,B 23.2416,C -1.1387,E1 23.1278,E2 240.9564} C_DIS
LIN {X -111.9263,Y -63.6284,Z 147,A -152.7387,B 23.2416,C -1.1412,E1 23.1296,E2 239.6411} C_DIS
LIN {X -109.5504,Y -67.6379,Z 147,A -150.6529,B 23.2417,C -1.1362,E1 23.1326,E2 237.5565} C_DIS
LIN {X -107.6914,Y -70.5597,Z 147,A -149.1237,B 23.242,C -1.1317,E1 23.1349,E2 236.0305} C_DIS
LIN {X -105.1215,Y -74.3339,Z 147,A -147.1041,B 23.2422,C -1.126,E1 23.1381,E2 234.0146} C_DIS
LIN {X -102.8869,Y -77.3974,Z 147,A -145.0495,B 23.2417,C -1.1381,E1 23.1416,E2 231.9184} C_DIS
LIN {X -100.4466,Y -80.5397,Z 147,A -143.5846,B 23.2425,C -1.1202,E1 23.1441,E2 230.4915} C_DIS
LIN {X -97.5508,Y -84.023,Z 147,A -141.6534,B 23.2429,C -1.1118,E1 23.1476,E2 228.5722} C_DIS
LIN {X -94.961,Y -86.9397,Z 147,A -139.8315,B 23.2429,C -1.1117,E1 23.151,E2 226.7419} C_DIS
LIN {X -91.752,Y -90.3198,Z 147,A -137.7748,B 23.2431,C -1.1064,E1 23.155,E2 224.6891} C_DIS
LIN {X -88.6693,Y -93.3485,Z 147,A -135.801,B 23.2431,C -1.1046,E1 23.1589,E2 222.7109} C_DIS
LIN {X -85.536,Y -96.2276,Z 147,A -133.8956,B 23.2433,C -1.1013,E1 23.1629,E2 220.8055} C_DIS
LIN {X -82.6832,Y -98.689,Z 147,A -132.2765,B 23.2436,C -1.0955,E1 23.1663,E2 219.1944} C_DIS
LIN {X -79.2635,Y -101.4566,Z 147,A -130.2682,B 23.2436,C -1.0941,E1 23.1707,E2 217.1815} C_DIS
LIN {X -76.0793,Y -103.8653,Z 147,A -128.1404,B 23.2431,C -1.1069,E1 23.1756,E2 215.0131} C_DIS
LIN {X -72.8428,Y -106.1601,Z 147,A -126.7355,B 23.2439,C -1.0876,E1 23.1787,E2 213.6521} C_DIS
LIN {X -70.1153,Y -107.9809,Z 147,A -125.0863,B 23.2437,C -1.0939,E1 23.1826,E2 211.9812} C_DIS
LIN {X -65.1617,Y -111.0405,Z 147,A -122.6717,B 23.2442,C -1.082,E1 23.1884,E2 209.5887} C_DIS
LIN {X -61.2815,Y -113.2288,Z 147,A -120.6287,B 23.2442,C -1.082,E1 23.1934,E2 207.5393} C_DIS
LIN {X -57.2515,Y -115.3166,Z 147,A -118.7252,B 23.2445,C -1.0742,E1 23.1981,E2 205.6501} C_DIS
LIN {X -54.2039,Y -116.7798,Z 147,A -116.9574,B 23.2441,C -1.0844,E1 23.2026,E2 203.8514} C_DIS
LIN {X -50.336,Y -118.5008,Z 147,A -115.1359,B 23.2443,C -1.0795,E1 23.2073,E2 202.0379} C_DIS
LIN {X -46.1429,Y -120.1944,Z 147,A -113.2709,B 23.2447,C -1.0707,E1 23.2121,E2 200.1908} C_DIS
LIN {X -42.704,Y -121.4589,Z 147,A -111.8088,B 23.2451,C -1.0615,E1 23.2159,E2 198.7489} C_DIS
LIN {X -38.702,Y -122.7924,Z 147,A -109.6947,B 23.2447,C -1.0709,E1 23.2216,E2 196.6068} C_DIS
LIN {X -35.165,Y -123.8518,Z 147,A -108.1331,B 23.2449,C -1.066,E1 23.2257,E2 195.0549} C_DIS
LIN {X -31.8739,Y -124.7385,Z 147,A -106.7369,B 23.2452,C -1.0595,E1 23.2294,E2 193.6729} C_DIS
LIN {X -29.2064,Y -125.391,Z 147,A -105.3483,B 23.2449,C -1.0666,E1 23.2333,E2 192.2644} C_DIS
LIN {X -24.8538,Y -126.3265,Z 147,A -103.4795,B 23.2451,C -1.0604,E1 23.2383,E2 190.4088} C_DIS
LIN {X -20.2901,Y -127.1389,Z 147,A -100.7552,B 23.2438,C -1.0908,E1 23.2461,E2 187.6046} C_DIS
LIN {X -15.5601,Y -127.8031,Z 147,A -99.4644,B 23.2455,C -1.0512,E1 23.2494,E2 186.4133} C_DIS
LIN {X -9.4723,Y -128.3976,Z 147,A -96.624,B 23.2453,C -1.0564,E1 23.2573,E2 183.558} C_DIS
LIN {X -4.4525,Y -128.6708,Z 147,A -94.1862,B 23.2449,C -1.066,E1 23.2642,E2 181.0954} C_DIS
LIN {X 0.9208,Y -128.7185,Z 147,A -92.2887,B 23.2459,C -1.0435,E1 23.2694,E2 179.2548} C_DIS
Enddeposition()
LIN {X 0.9208,Y -128.7185,Z 147,A -92.2887,B 23.2459,C -1.0435,E1 23.2694,E2 179.2548} C_DIS
Startdeposition()
$VEL.CP = VEL_PRINT
LIN {X -0.9065,Y -127.7891,Z 147,A -93.0891,B 22.3667,C -0.8975,E1 22.3821,E2 180.3236} C_DIS
LIN {X -7.4127,Y -127.5776,Z 147,A -95.9372,B 22.3665,C -0.9003,E1 22.3742,E2 183.1649} C_DIS
LIN {X -11.6535,Y -127.2608,Z 147,A -98.0424,B 22.3669,C -0.8917,E1 22.3682,E2 185.294} C_DIS
LIN {X -15.2054,Y -126.8841,Z 147,A -100.0257,B 22.3675,C -0.8752,E1 22.3626,E2 187.3221} C_DIS
LIN {X -19.1842,Y -126.3443,Z 147,A -101.176,B 22.3664,C -0.9041,E1 22.3596,E2 188.3974} C_DIS
LIN {X -23.7518,Y -125.5654,Z 147,A -103.2051,B 22.3663,C -0.9069,E1 22.3541,E2 190.4212} C_DIS
LIN {X -26.8983,Y -124.9289,Z 147,A -104.8986,B 22.3667,C -0.8964,E1 22.3493,E2 192.1447} C_DIS
LIN {X -30.6605,Y -124.0613,Z 147,A -106.726,B 22.3668,C -0.8932,E1 22.3443,E2 193.9835} C_DIS
LIN {X -34.6497,Y -123.0048,Z 147,A -108.4319,B 22.3665,C -0.9006,E1 22.3398,E2 195.6726} C_DIS
LIN {X -37.9,Y -122.0434,Z 147,A -110.0122,B 22.3665,C -0.8991,E1 22.3356,E2 197.2601} C_DIS
LIN {X -42.6975,Y -120.4495,Z 147,A -112.2137,B 22.3665,C -0.9038,E1 22.3298,E2 199.4539} C_DIS
LIN {X -46.037,Y -119.2115,Z 147,A -114.0739,B 22.3668,C -0.894,E1 22.3248,E2 201.3443} C_DIS
LIN {X -50.3017,Y -117.4761,Z 147,A -116.1488,B 22.3668,C -0.8957,E1 22.3195,E2 203.4201} C_DIS
LIN {X -55.1402,Y -115.2833,Z 147,A -118.3438,B 22.3663,C -0.9064,E1 22.314,E2 205.593} C_DIS
LIN {X -58.3375,Y -113.6995,Z 147,A -119.953,B 22.3663,C -0.908,E1 22.3099,E2 207.2028} C_DIS
LIN {X -62.0232,Y -111.7332,Z 147,A -121.8883,B 22.3663,C -0.9079,E1 22.3052,E2 209.1447} C_DIS
LIN {X -65.8923,Y -109.4963,Z 147,A -123.7411,B 22.3659,C -0.9172,E1 22.3008,E2 210.9793} C_DIS
LIN {X -69.1217,Y -107.4869,Z 147,A -125.3827,B 22.3657,C -0.9225,E1 22.2969,E2 212.6127} C_DIS
LIN {X -71.6384,Y -105.8258,Z 147,A -127.0449,B 22.3661,C -0.9116,E1 22.293,E2 214.3101} C_DIS
LIN {X -76.6484,Y -102.2563,Z 147,A -129.5859,B 22.3656,C -0.9254,E1 22.2873,E2 216.8245} C_DIS
LIN {X -79.3309,Y -100.1892,Z 147,A -131.3115,B 22.3658,C -0.9195,E1 22.2834,E2 218.573} C_DIS
LIN {X -82.5096,Y -97.5881,Z 147,A -133.1584,B 22.3657,C -0.9227,E1 22.2795,E2 220.4193} C_DIS
LIN {X -85.7753,Y -94.73,Z 147,A -135.0875,B 22.3655,C -0.9273,E1 22.2754,E2 222.345} C_DIS
LIN {X -89.1112,Y -91.5994,Z 147,A -137.154,B 22.3654,C -0.9309,E1 22.2713,E2 224.4118} C_DIS
LIN {X -92.1751,Y -88.5156,Z 147,A -139.101,B 22.3652,C -0.9352,E1 22.2675,E2 226.3569} C_DIS
LIN {X -95.0927,Y -85.3731,Z 147,A -141.0369,B 22.365,C -0.9389,E1 22.2638,E2 228.2927} C_DIS
LIN {X -98.0279,Y -81.9862,Z 147,A -143.0514,B 22.3649,C -0.9433,E1 22.2602,E2 230.3058} C_DIS
LIN {X -100.9917,Y -78.3056,Z 147,A -145.4358,B 22.3651,C -0.9375,E1 22.256,E2 232.7185} C_DIS
LIN {X -103.0523,Y -75.5739,Z 147,A -146.399,B 22.364,C -0.9648,E1 22.2545,E2 233.6147} C_DIS
LIN {X -105.9327,Y -71.4802,Z 147,A -148.8785,B 22.3642,C -0.9607,E1 22.2505,E2 236.1189} C_DIS
LIN {X -108.0698,Y -68.2061,Z 147,A -150.6577,B 22.364,C -0.9641,E1 22.2478,E2 237.8991} C_DIS
LIN {X -110.0654,Y -64.9371,Z 147,A -152.4743,B 22.364,C -0.9646,E1 22.2452,E2 239.7251} C_DIS
LIN {X -111.6856,Y -62.1092,Z 147,A -153.8764,B 22.3637,C -0.971,E1 22.2433,E2 241.1188} C_DIS
LIN {X -113.9223,Y -57.8998,Z 147,A -156.0057,B 22.3635,C -0.9772,E1 22.2405,E2 243.2445} C_DIS
LIN {X -115.4261,Y -54.8414,Z 147,A -157.5255,B 22.3633,C -0.9818,E1 22.2387,E2 244.7614} C_DIS
LIN {X -116.8892,Y -51.652,Z 147,A -159.0863,B 22.3631,C -0.9868,E1 22.2369,E2 246.3188} C_DIS
LIN {X -118.1654,Y -48.6625,Z 147,A -160.5754,B 22.363,C -0.9896,E1 22.2353,E2 247.8096} C_DIS
LIN {X -119.2634,Y -45.9035,Z 147,A -161.9004,B 22.3628,C -0.9938,E1 22.2339,E2 249.132} C_DIS
LIN {X -121.4454,Y -39.776,Z 147,A -164.8834,B 22.3625,C -0.9997,E1 22.2312,E2 252.1186} C_DIS
LIN {X -122.8772,Y -35.1005,Z 147,A -167.3547,B 22.3627,C -0.995,E1 22.2292,E2 254.6185} C_DIS
LIN {X -124.2123,Y -30.034,Z 147,A -169.4947,B 22.3621,C -1.0107,E1 22.2278,E2 256.7312} C_DIS
LIN {X -125.1045,Y -26.0763,Z 147,A -171.3714,B 22.3619,C -1.0139,E1 22.2266,E2 258.6117} C_DIS
LIN {X -125.7985,Y -22.483,Z 147,A -172.9716,B 22.3616,C -1.0207,E1 22.2258,E2 260.2048} C_DIS
LIN {X -126.4577,Y -18.4215,Z 147,A -174.8099,B 22.3614,C -1.0268,E1 22.2251,E2 262.0395} C_DIS
LIN {X -126.9065,Y -15.0175,Z 147,A -176.349,B 22.3612,C -1.0316,E1 22.2245,E2 263.5761} C_DIS
LIN {X -127.3192,Y -10.9852,Z 147,A -178.1979,B 22.361,C -1.0361,E1 22.224,E2 265.4257} C_DIS
LIN {X -127.5545,Y -7.7881,Z 147,A -179.6227,B 22.3607,C -1.0412,E1 22.2238,E2 266.8467} C_DIS
LIN {X -127.7291,Y -4.0416,Z 147,A 178.6393,B 22.3607,C -1.0443,E1 22.2236,E2 268.5885} C_DIS
LIN {X -127.793,Y -0.4134,Z 147,A 176.9727,B 22.3604,C -1.0479,E1 22.2236,E2 270.2569} C_DIS
LIN {X -127.7435,Y 3.5233,Z 147,A 175.2362,B 22.3601,C -1.0547,E1 22.2236,E2 271.9872} C_DIS
LIN {X -127.5671,Y 7.5845,Z 147,A 173.4154,B 22.3599,C -1.0606,E1 22.2239,E2 273.8048} C_DIS
LIN {X -127.3102,Y 11.0913,Z 147,A 171.855,B 22.3596,C -1.0663,E1 22.2242,E2 275.3607} C_DIS
LIN {X -126.8931,Y 15.1302,Z 147,A 169.9538,B 22.3596,C -1.0689,E1 22.2248,E2 277.2679} C_DIS
LIN {X -126.3147,Y 19.3749,Z 147,A 168.028,B 22.3592,C -1.0749,E1 22.2256,E2 279.191} C_DIS
LIN {X -125.7432,Y 22.792,Z 147,A 166.4185,B 22.3592,C -1.0776,E1 22.2263,E2 280.8043} C_DIS
LIN {X -124.8821,Y 27.1151,Z 147,A 164.5509,B 22.3586,C -1.0882,E1 22.2274,E2 282.6562} C_DIS
LIN {X -124.1352,Y 30.3541,Z 147,A 162.8804,B 22.3587,C -1.0857,E1 22.2285,E2 284.3444} C_DIS
LIN {X -121.6696,Y 39.0801,Z 147,A 158.8967,B 22.358,C -1.1017,E1 22.2316,E2 288.312} C_DIS
LIN {X -119.1565,Y 46.1785,Z 147,A 155.5066,B 22.3575,C -1.1115,E1 22.2348,E2 291.6978} C_DIS
LIN {X -117.928,Y 49.2309,Z 147,A 154.0197,B 22.3573,C -1.1155,E1 22.2364,E2 293.1836} C_DIS
LIN {X -116.5579,Y 52.3928,Z 147,A 152.4393,B 22.3572,C -1.1187,E1 22.2381,E2 294.7653} C_DIS
LIN {X -113.5026,Y 58.7233,Z 147,A 149.3287,B 22.3567,C -1.1296,E1 22.242,E2 297.8661} C_DIS
LIN {X -111.9716,Y 61.5926,Z 147,A 147.7538,B 22.3567,C -1.1291,E1 22.2441,E2 299.4518} C_DIS
LIN {X -107.8961,Y 68.4814,Z 147,A 144.3229,B 22.3559,C -1.1456,E1 22.249,E2 302.8588} C_DIS
LIN {X -106.0924,Y 71.244,Z 147,A 142.6311,B 22.3561,C -1.1411,E1 22.2516,E2 304.5722} C_DIS
LIN {X -103.0001,Y 75.6449,Z 147,A 140.2166,B 22.3558,C -1.1475,E1 22.2555,E2 306.9831} C_DIS
LIN {X -99.5417,Y 80.1413,Z 147,A 137.6411,B 22.3555,C -1.1529,E1 22.2599,E2 309.5582} C_DIS
LIN {X -96.3811,Y 83.9158,Z 147,A 135.2691,B 22.3555,C -1.1518,E1 22.2643,E2 311.9453} C_DIS
LIN {X -92.9437,Y 87.7077,Z 147,A 133.1202,B 22.355,C -1.1635,E1 22.2683,E2 314.0742} C_DIS
LIN {X -89.834,Y 90.8908,Z 147,A 131.0568,B 22.355,C -1.1654,E1 22.2724,E2 316.1423} C_DIS
LIN {X -86.1969,Y 94.3472,Z 147,A 128.823,B 22.3546,C -1.1713,E1 22.2769,E2 318.371} C_DIS
LIN {X -82.9401,Y 97.2222,Z 147,A 126.8831,B 22.3544,C -1.176,E1 22.281,E2 320.3071} C_DIS
LIN {X -79.5428,Y 100.0205,Z 147,A 124.6187,B 22.3548,C -1.1683,E1 22.286,E2 322.6015} C_DIS
LIN {X -76.6905,Y 102.2241,Z 147,A 123.3542,B 22.3539,C -1.186,E1 22.2887,E2 323.8242} C_DIS
LIN {X -73.4002,Y 104.6119,Z 147,A 121.4351,B 22.3539,C -1.1857,E1 22.2931,E2 325.7516} C_DIS
LIN {X -69.8087,Y 107.042,Z 147,A 119.4818,B 22.3537,C -1.1891,E1 22.2976,E2 327.7035} C_DIS
LIN {X -65.7305,Y 109.5938,Z 147,A 116.5744,B 22.3551,C -1.1621,E1 22.3048,E2 330.6921} C_DIS
LIN {X -60.6042,Y 112.5091,Z 147,A 114.6052,B 22.3535,C -1.1944,E1 22.3094,E2 332.5826} C_DIS
LIN {X -57.6897,Y 114.0292,Z 147,A 113.2573,B 22.3531,C -1.202,E1 22.3127,E2 333.9144} C_DIS
LIN {X -53.3495,Y 116.1232,Z 147,A 111.1559,B 22.3528,C -1.2078,E1 22.318,E2 336.0066} C_DIS
LIN {X -50.3704,Y 117.4464,Z 147,A 109.6254,B 22.3528,C -1.207,E1 22.3219,E2 337.5433} C_DIS
LIN {X -46.4496,Y 119.0511,Z 147,A 107.7555,B 22.3526,C -1.2108,E1 22.3268,E2 339.4078} C_DIS
LIN {X -43.3605,Y 120.2105,Z 147,A 106.2953,B 22.3526,C -1.2135,E1 22.3306,E2 340.8644} C_DIS
LIN {X -39.5,Y 121.5348,Z 147,A 104.2404,B 22.3529,C -1.2061,E1 22.3361,E2 342.9429} C_DIS
LIN {X -34.7691,Y 122.9714,Z 147,A 102.1679,B 22.3524,C -1.2146,E1 22.3416,E2 344.997} C_DIS
LIN {X -31.2528,Y 123.9114,Z 147,A 100.5491,B 22.3524,C -1.2167,E1 22.346,E2 346.6128} C_DIS
LIN {X -27.1703,Y 124.8702,Z 147,A 98.6799,B 22.3522,C -1.2189,E1 22.351,E2 348.4792} C_DIS
LIN {X -23.7201,Y 125.5715,Z 147,A 96.8518,B 22.3527,C -1.2095,E1 22.3561,E2 350.3343} C_DIS
LIN {X -18.8625,Y 126.3941,Z 147,A 94.944,B 22.352,C -1.2238,E1 22.3613,E2 352.2064} C_DIS
LIN {X -15.5952,Y 126.8376,Z 147,A 93.33,B 22.3522,C -1.2188,E1 22.3658,E2 353.8348} C_DIS
LIN {X -9.5626,Y 127.434,Z 147,A 90.6498,B 22.3521,C -1.2217,E1 22.3732,E2 356.5089} C_DIS
LIN {X -3.6773,Y 127.7392,Z 147,A 88.0219,B 22.3521,C -1.2231,E1 22.3806,E2 359.1336} C_DIS
LIN {X 0.102,Y 127.7935,Z 147,A 85.9399,B 22.3528,C -1.2067,E1 22.3865,E2 361.2587} C_DIS
LIN {X 3.7794,Y 127.7364,Z 147,A 84.5317,B 22.3523,C -1.2173,E1 22.3903,E2 362.6389} C_DIS
LIN {X 8.5973,Y 127.5045,Z 147,A 82.4469,B 22.3521,C -1.2206,E1 22.3961,E2 364.7141} C_DIS
LIN {X 12.5665,Y 127.1731,Z 147,A 80.4732,B 22.3526,C -1.2122,E1 22.4017,E2 366.7085} C_DIS
LIN {X 17.7957,Y 126.5471,Z 147,A 78.2153,B 22.3524,C -1.2161,E1 22.4079,E2 368.954} C_DIS
LIN {X 21.7499,Y 125.9295,Z 147,A 76.4501,B 22.3524,C -1.2167,E1 22.4127,E2 370.7156} C_DIS
LIN {X 25.6418,Y 125.1929,Z 147,A 74.7398,B 22.3522,C -1.2188,E1 22.4174,E2 372.418} C_DIS
LIN {X 29.7316,Y 124.2852,Z 147,A 72.9291,B 22.3522,C -1.2208,E1 22.4223,E2 374.2207} C_DIS
LIN {X 33.0045,Y 123.4562,Z 147,A 71.448,B 22.3521,C -1.2213,E1 22.4263,E2 375.6981} C_DIS
LIN {X 36.1155,Y 122.5824,Z 147,A 70.0008,B 22.3521,C -1.2203,E1 22.4302,E2 377.1451} C_DIS
LIN {X 40.1353,Y 121.3257,Z 147,A 68.3287,B 22.3517,C -1.2284,E1 22.4346,E2 378.7924} C_DIS
LIN {X 43.0844,Y 120.3101,Z 147,A 66.5741,B 22.3526,C -1.2113,E1 22.4393,E2 380.5879} C_DIS
LIN {X 46.8684,Y 118.8883,Z 147,A 64.6861,B 22.3529,C -1.2061,E1 22.4442,E2 382.4848} C_DIS
LIN {X 51.0122,Y 117.1689,Z 147,A 62.9701,B 22.3523,C -1.2171,E1 22.4486,E2 384.1673} C_DIS
LIN {X 53.8304,Y 115.9009,Z 147,A 61.5948,B 22.3523,C -1.2159,E1 22.4521,E2 385.5418} C_DIS
LIN {X 56.6187,Y 114.5644,Z 147,A 60.1303,B 22.3526,C -1.2107,E1 22.4558,E2 387.0156} C_DIS
LIN {X 59.628,Y 113.0276,Z 147,A 58.6759,B 22.3526,C -1.2114,E1 22.4594,E2 388.4636} C_DIS
LIN {X 64.1641,Y 110.5177,Z 147,A 56.0586,B 22.3535,C -1.1949,E1 22.4658,E2 391.1154} C_DIS
LIN {X 67.7092,Y 108.3821,Z 147,A 54.3689,B 22.3532,C -1.1995,E1 22.4698,E2 392.7869} C_DIS
LIN {X 71.3688,Y 106.0084,Z 147,A 52.3994,B 22.3534,C -1.1957,E1 22.4744,E2 394.759} C_DIS
LIN {X 74.8988,Y 103.544,Z 147,A 50.5064,B 22.3534,C -1.1941,E1 22.4787,E2 396.6488} C_DIS
LIN {X 78.2751,Y 101.0157,Z 147,A 48.6276,B 22.3536,C -1.1912,E1 22.4828,E2 398.5273} C_DIS
LIN {X 81.74,Y 98.2335,Z 147,A 46.6364,B 22.3538,C -1.1875,E1 22.4872,E2 400.5197} C_DIS
LIN {X 84.9829,Y 95.4422,Z 147,A 44.7179,B 22.354,C -1.1837,E1 22.4912,E2 402.4396} C_DIS
LIN {X 88.5503,Y 92.1419,Z 147,A 42.5767,B 22.3542,C -1.1809,E1 22.4955,E2 404.5781} C_DIS
LIN {X 90.9776,Y 89.7461,Z 147,A 40.7239,B 22.3551,C -1.1628,E1 22.4993,E2 406.4693} C_DIS
LIN {X 93.5169,Y 87.0962,Z 147,A 39.6105,B 22.354,C -1.1836,E1 22.5013,E2 407.5229} C_DIS
LIN {X 95.8184,Y 84.5578,Z 147,A 37.8719,B 22.3547,C -1.1707,E1 22.5046,E2 409.2863} C_DIS
LIN {X 98.6479,Y 81.2396,Z 147,A 35.926,B 22.3549,C -1.1666,E1 22.5081,E2 411.233} C_DIS
LIN {X 101.3276,Y 77.8715,Z 147,A 33.9949,B 22.3551,C -1.1619,E1 22.5114,E2 413.1661} C_DIS
LIN {X 103.9262,Y 74.3674,Z 147,A 32.0549,B 22.3553,C -1.1577,E1 22.5146,E2 415.1064} C_DIS
LIN {X 106.4941,Y 70.6421,Z 147,A 30.0472,B 22.3555,C -1.1535,E1 22.5177,E2 417.1138} C_DIS
LIN {X 108.7519,Y 67.1133,Z 147,A 28.2146,B 22.3556,C -1.1507,E1 22.5204,E2 418.9433} C_DIS
LIN {X 110.3259,Y 64.4938,Z 147,A 26.8055,B 22.3559,C -1.1452,E1 22.5224,E2 420.3585} C_DIS
LIN {X 112.3946,Y 60.8175,Z 147,A 24.9487,B 22.3561,C -1.1417,E1 22.525,E2 422.2135} C_DIS
Enddeposition()
END
